C09142=1184.403,208.297,-60.136,-177.705,6.782,148.579
C09143=1184.398,208.546,-60.161,-177.703,6.784,148.579
C09144=1184.394,208.794,-60.185,-177.700,6.786,148.579
C09145=1184.389,209.044,-60.210,-177.698,6.788,148.579
C09146=1184.385,209.292,-60.234,-177.695,6.790,148.578
C09147=1184.381,209.541,-60.258,-177.692,6.792,148.578
C09148=1184.376,209.790,-60.283,-177.690,6.794,148.578
C09149=1184.372,210.039,-60.307,-177.687,6.796,148.577
C09150=1184.366,210.309,-60.333,-177.684,6.799,148.577
C09151=1184.361,210.579,-60.360,-177.681,6.801,148.577
C09152=1184.357,210.850,-60.387,-177.678,6.803,148.576
C09153=1184.351,211.121,-60.414,-177.675,6.806,148.576
C09154=1184.347,211.369,-60.438,-177.673,6.808,148.576
C09155=1184.342,211.618,-60.463,-177.670,6.810,148.576
C09156=1184.338,211.867,-60.487,-177.667,6.812,148.575
C09157=1184.333,212.116,-60.512,-177.665,6.815,148.575
C09158=1184.329,212.365,-60.536,-177.662,6.816,148.575
C09159=1184.324,212.613,-60.561,-177.659,6.818,148.575
C09160=1184.320,212.861,-60.586,-177.657,6.821,148.575
C09161=1184.315,213.111,-60.611,-177.654,6.823,148.574
C09162=1184.310,213.359,-60.635,-177.651,6.825,148.574
C09163=1184.306,213.608,-60.659,-177.649,6.827,148.574
C09164=1184.301,213.857,-60.684,-177.646,6.830,148.573
C09165=1184.297,214.106,-60.708,-177.643,6.831,148.573
C09166=1184.293,214.354,-60.734,-177.640,6.833,148.573
C09167=1184.288,214.603,-60.758,-177.638,6.835,148.573
C09168=1184.283,214.851,-60.783,-177.635,6.838,148.572
C09169=1184.279,215.101,-60.808,-177.632,6.840,148.572
C09170=1184.275,215.349,-60.833,-177.630,6.842,148.572
C09171=1184.270,215.598,-60.858,-177.627,6.845,148.572
C09172=1184.266,215.847,-60.882,-177.624,6.846,148.571
C09173=1184.260,216.095,-60.907,-177.622,6.848,148.571
C09174=1184.256,216.344,-60.932,-177.620,6.850,148.571
C09175=1184.252,216.592,-60.956,-177.616,6.853,148.570
C09176=1184.247,216.842,-60.981,-177.614,6.855,148.570
C09177=1184.243,217.090,-61.007,-177.611,6.857,148.570
C09178=1184.239,217.339,-61.031,-177.608,6.859,148.570
C09179=1184.234,217.588,-61.056,-177.606,6.862,148.570
C09180=1184.229,217.836,-61.081,-177.603,6.863,148.569
C09181=1184.225,218.085,-61.106,-177.601,6.866,148.569
C09182=1184.220,218.334,-61.130,-177.598,6.868,148.569
C09183=1184.216,218.583,-61.156,-177.595,6.870,148.569
C09184=1184.210,218.831,-61.181,-177.593,6.873,148.568
C09185=1184.207,219.080,-61.206,-177.590,6.875,148.568
C09186=1184.202,219.329,-61.231,-177.587,6.877,148.568
C09187=1184.198,219.577,-61.256,-177.585,6.879,148.568
C09188=1184.192,219.826,-61.281,-177.582,6.881,148.567
C09189=1184.189,220.075,-61.306,-177.579,6.883,148.567
C09190=1184.184,220.323,-61.331,-177.577,6.885,148.567
C09191=1184.180,220.572,-61.357,-177.574,6.888,148.567
C09192=1184.175,220.821,-61.381,-177.572,6.890,148.566
C09193=1184.171,221.069,-61.406,-177.569,6.892,148.566
C09194=1184.166,221.318,-61.431,-177.566,6.895,148.566
C09195=1184.162,221.567,-61.457,-177.564,6.897,148.566
C09196=1184.157,221.816,-61.482,-177.561,6.899,148.565
C09197=1184.152,222.064,-61.507,-177.558,6.901,148.565
C09198=1184.147,222.313,-61.532,-177.556,6.903,148.565
C09199=1184.144,222.562,-61.557,-177.553,6.905,148.565
C09200=1184.139,222.810,-61.583,-177.550,6.908,148.565
C09201=1184.134,223.059,-61.608,-177.548,6.910,148.564
C09202=1184.130,223.308,-61.633,-177.545,6.912,148.564
C09203=1184.125,223.557,-61.658,-177.542,6.915,148.564
C09204=1184.121,223.805,-61.684,-177.539,6.916,148.564
C09205=1184.116,224.054,-61.709,-177.537,6.919,148.563
C09206=1184.111,224.303,-61.734,-177.534,6.921,148.563
C09207=1184.107,224.551,-61.759,-177.531,6.923,148.563
C09208=1184.103,224.800,-61.785,-177.529,6.925,148.563
C09209=1184.099,225.048,-61.810,-177.526,6.928,148.562
C09210=1184.094,225.297,-61.835,-177.524,6.930,148.562
C09211=1184.090,225.546,-61.861,-177.521,6.932,148.562
C09212=1184.085,225.794,-61.886,-177.518,6.935,148.562
C09213=1184.080,226.043,-61.911,-177.516,6.937,148.562
C09214=1184.076,226.292,-61.937,-177.513,6.939,148.561
C09215=1184.071,226.540,-61.962,-177.510,6.941,148.561
C09216=1184.067,226.789,-61.988,-177.508,6.943,148.561
C09217=1184.063,227.038,-62.014,-177.505,6.946,148.561
C09218=1184.058,227.287,-62.039,-177.502,6.948,148.560
C09219=1184.053,227.535,-62.064,-177.500,6.950,148.560
C09220=1184.048,227.784,-62.090,-177.497,6.953,148.560
C09221=1184.044,228.032,-62.116,-177.494,6.955,148.560
C09222=1184.040,228.281,-62.141,-177.492,6.957,148.560
C09223=1184.035,228.529,-62.167,-177.489,6.959,148.559
C09224=1184.031,228.778,-62.192,-177.487,6.961,148.559
C09225=1184.027,229.027,-62.218,-177.484,6.964,148.559
C09226=1184.022,229.276,-62.243,-177.481,6.966,148.559
C09227=1184.017,229.524,-62.269,-177.479,6.968,148.558
C09228=1184.013,229.773,-62.294,-177.476,6.971,148.558
C09229=1184.008,230.021,-62.320,-177.473,6.973,148.558
C09230=1184.004,230.270,-62.345,-177.471,6.975,148.558
C09231=1183.999,230.519,-62.372,-177.468,6.978,148.558
C09232=1183.995,230.768,-62.398,-177.465,6.979,148.557
C09233=1183.990,231.016,-62.423,-177.463,6.982,148.557
C09234=1183.986,231.265,-62.449,-177.460,6.984,148.557
C09235=1183.982,231.514,-62.474,-177.458,6.986,148.557
C09236=1183.977,231.762,-62.500,-177.454,6.989,148.556
C09237=1183.973,232.011,-62.526,-177.452,6.991,148.556
C09238=1183.968,232.259,-62.551,-177.449,6.994,148.556
C09239=1183.963,232.509,-62.578,-177.447,6.996,148.556
C09240=1183.959,232.756,-62.604,-177.444,6.998,148.556
C09241=1183.955,233.005,-62.630,-177.442,7.001,148.556
C09242=1183.950,233.254,-62.655,-177.439,7.003,148.555
C09243=1183.946,233.502,-62.681,-177.436,7.006,148.555
C09244=1183.941,233.751,-62.707,-177.434,7.007,148.555
C09245=1183.936,234.000,-62.733,-177.431,7.009,148.555
C09246=1183.932,234.249,-62.758,-177.428,7.012,148.554
C09247=1183.928,234.497,-62.784,-177.426,7.014,148.554
C09248=1183.923,234.745,-62.810,-177.423,7.017,148.554
C09249=1183.919,234.994,-62.837,-177.421,7.019,148.554
C09250=1183.914,235.243,-62.862,-177.418,7.021,148.554
C09251=1183.910,235.492,-62.888,-177.415,7.024,148.554
C09252=1183.906,235.740,-62.914,-177.413,7.026,148.553
C09253=1183.901,235.988,-62.941,-177.410,7.029,148.553
C09254=1183.896,236.260,-62.969,-177.407,7.031,148.553
C09255=1183.891,236.531,-62.997,-177.404,7.033,148.553
C09256=1183.886,236.804,-63.026,-177.401,7.036,148.552
C09257=1183.882,237.075,-63.055,-177.398,7.039,148.552
C09258=1183.877,237.323,-63.080,-177.396,7.041,148.552
C09259=1183.873,237.572,-63.106,-177.393,7.044,148.552
C09260=1183.868,237.820,-63.133,-177.390,7.046,148.552
C09261=1183.864,238.069,-63.159,-177.388,7.048,148.552
C09262=1183.860,238.318,-63.185,-177.385,7.050,148.551
C09263=1183.855,238.566,-63.212,-177.383,7.053,148.551
C09264=1183.851,238.815,-63.237,-177.380,7.055,148.551
C09265=1183.845,239.064,-63.263,-177.377,7.057,148.551
C09266=1183.841,239.312,-63.290,-177.375,7.060,148.551
C09267=1183.837,239.561,-63.316,-177.372,7.062,148.550
C09268=1183.832,239.809,-63.343,-177.369,7.065,148.550
C09269=1183.828,240.058,-63.368,-177.367,7.067,148.550
C09270=1183.823,240.306,-63.395,-177.364,7.070,148.550
C09271=1183.819,240.555,-63.421,-177.361,7.072,148.550
C09272=1183.815,240.804,-63.447,-177.359,7.074,148.550
C09273=1183.810,241.052,-63.474,-177.356,7.077,148.549
C09274=1183.805,241.301,-63.499,-177.354,7.079,148.549
C09275=1183.801,241.549,-63.526,-177.351,7.082,148.549
C09276=1183.797,241.798,-63.552,-177.348,7.084,148.549
C09277=1183.792,242.046,-63.579,-177.346,7.087,148.549
C09278=1183.788,242.294,-63.606,-177.343,7.088,148.548
C09279=1183.783,242.544,-63.632,-177.340,7.091,148.548
C09280=1183.779,242.792,-63.659,-177.338,7.093,148.548
C09281=1183.774,243.041,-63.685,-177.335,7.096,148.548
C09282=1183.770,243.289,-63.711,-177.333,7.098,148.548
C09283=1183.765,243.538,-63.738,-177.330,7.101,148.548
C09284=1183.761,243.786,-63.764,-177.327,7.103,148.547
C09285=1183.757,244.035,-63.791,-177.325,7.106,148.547
C09286=1183.752,244.284,-63.817,-177.322,7.108,148.547
C09287=1183.748,244.532,-63.844,-177.319,7.111,148.547
C09288=1183.744,244.780,-63.870,-177.317,7.113,148.547
C09289=1183.739,245.030,-63.897,-177.314,7.115,148.547
C09290=1183.735,245.278,-63.923,-177.312,7.118,148.547
C09291=1183.730,245.526,-63.950,-177.309,7.120,148.546
C09292=1183.726,245.775,-63.977,-177.306,7.123,148.546
C09293=1183.721,246.023,-64.003,-177.304,7.125,148.546
C09294=1183.717,246.272,-64.030,-177.301,7.127,148.546
C09295=1183.713,246.520,-64.057,-177.299,7.130,148.546
C09296=1183.708,246.769,-64.084,-177.296,7.132,148.546
C09297=1183.703,247.018,-64.110,-177.293,7.134,148.545
C09298=1183.699,247.266,-64.137,-177.291,7.137,148.545
C09299=1183.695,247.514,-64.164,-177.288,7.139,148.545
C09300=1183.690,247.763,-64.191,-177.285,7.142,148.545
C09301=1183.686,248.011,-64.217,-177.283,7.144,148.545
C09302=1183.681,248.260,-64.243,-177.280,7.147,148.545
C09303=1183.677,248.509,-64.271,-177.278,7.149,148.544
C09304=1183.673,248.757,-64.297,-177.275,7.152,148.544
C09305=1183.668,249.005,-64.324,-177.272,7.155,148.544
C09306=1183.663,249.254,-64.351,-177.270,7.157,148.544
C09307=1183.659,249.502,-64.378,-177.267,7.160,148.544
C09308=1183.655,249.751,-64.405,-177.264,7.162,148.544
C09309=1183.650,249.999,-64.432,-177.261,7.165,148.544
C09310=1183.646,250.247,-64.458,-177.259,7.167,148.543
C09311=1183.642,250.497,-64.485,-177.256,7.169,148.543
C09312=1183.637,250.746,-64.512,-177.254,7.172,148.543
C09313=1183.632,250.994,-64.539,-177.251,7.175,148.543
C09314=1183.629,251.242,-64.566,-177.249,7.176,148.543
C09315=1183.624,251.491,-64.593,-177.246,7.179,148.543
C09316=1183.619,251.739,-64.620,-177.244,7.182,148.543
C09317=1183.615,251.988,-64.647,-177.241,7.184,148.542
C09318=1183.610,252.236,-64.674,-177.238,7.186,148.542
C09319=1183.607,252.485,-64.701,-177.236,7.189,148.542
C09320=1183.602,252.733,-64.728,-177.233,7.191,148.542
C09321=1183.598,252.982,-64.755,-177.230,7.194,148.542
C09322=1183.593,253.230,-64.782,-177.227,7.197,148.542
C09323=1183.588,253.479,-64.810,-177.225,7.199,148.542
C09324=1183.584,253.727,-64.837,-177.222,7.202,148.541
C09325=1183.580,253.975,-64.863,-177.220,7.204,148.541
C09326=1183.576,254.224,-64.890,-177.217,7.207,148.541
C09327=1183.571,254.473,-64.918,-177.215,7.209,148.541
C09328=1183.567,254.721,-64.945,-177.212,7.212,148.541
C09329=1183.562,254.969,-64.972,-177.210,7.214,148.541
C09330=1183.557,255.218,-64.999,-177.207,7.217,148.541
C09331=1183.553,255.466,-65.027,-177.204,7.220,148.541
C09332=1183.549,255.715,-65.054,-177.202,7.222,148.540
C09333=1183.544,255.963,-65.082,-177.199,7.225,148.540
C09334=1183.540,256.211,-65.108,-177.197,7.227,148.540
C09335=1183.536,256.460,-65.135,-177.193,7.230,148.540
C09336=1183.532,256.709,-65.163,-177.191,7.232,148.540
C09337=1183.527,256.957,-65.190,-177.189,7.235,148.540
C09338=1183.523,257.206,-65.218,-177.186,7.238,148.540
C09339=1183.518,257.454,-65.245,-177.183,7.240,148.539
C09340=1183.513,257.703,-65.272,-177.180,7.242,148.539
C09341=1183.510,257.951,-65.300,-177.178,7.245,148.539
C09342=1183.505,258.200,-65.327,-177.176,7.248,148.539
C09343=1183.500,258.448,-65.354,-177.173,7.249,148.539
C09344=1183.496,258.696,-65.382,-177.170,7.252,148.539
C09345=1183.492,258.945,-65.409,-177.167,7.255,148.539
C09346=1183.487,259.193,-65.437,-177.165,7.258,148.539
C09347=1183.483,259.442,-65.464,-177.163,7.261,148.539
C09348=1183.479,259.691,-65.491,-177.160,7.262,148.538
C09349=1183.474,259.939,-65.519,-177.157,7.265,148.538
C09350=1183.470,260.187,-65.546,-177.154,7.268,148.538
C09351=1183.465,260.435,-65.574,-177.152,7.270,148.538
C09352=1183.461,260.685,-65.602,-177.149,7.273,148.538
C09353=1183.456,260.932,-65.630,-177.147,7.275,148.538
C09354=1183.452,261.181,-65.657,-177.144,7.278,148.538
C09355=1183.448,261.429,-65.685,-177.141,7.281,148.538
C09356=1183.443,261.678,-65.712,-177.139,7.283,148.538
C09357=1183.439,261.926,-65.740,-177.136,7.286,148.537
C09358=1183.434,262.199,-65.771,-177.133,7.289,148.537
C09359=1183.429,262.472,-65.801,-177.131,7.292,148.537
C09360=1183.425,262.745,-65.831,-177.127,7.295,148.537
C09361=1183.420,263.017,-65.861,-177.125,7.298,148.537
C09362=1183.416,263.267,-65.889,-177.123,7.300,148.537
C09363=1183.411,263.515,-65.917,-177.120,7.303,148.537
C09364=1183.406,263.763,-65.944,-177.117,7.305,148.536
C09365=1183.402,264.012,-65.972,-177.114,7.308,148.536
C09366=1183.398,264.260,-66.000,-177.112,7.311,148.536
C09367=1183.394,264.509,-66.027,-177.110,7.313,148.536
C09368=1183.389,264.757,-66.056,-177.107,7.316,148.536
C09369=1183.384,265.005,-66.084,-177.104,7.319,148.536
C09370=1183.380,265.254,-66.111,-177.101,7.321,148.536
C09371=1183.376,265.502,-66.139,-177.099,7.324,148.536
C09372=1183.372,265.750,-66.167,-177.096,7.327,148.536
C09373=1183.367,265.999,-66.195,-177.094,7.329,148.536
C09374=1183.362,266.247,-66.222,-177.091,7.332,148.536
C09375=1183.359,266.496,-66.250,-177.089,7.334,148.536
C09376=1183.354,266.744,-66.279,-177.086,7.337,148.535
C09377=1183.349,266.992,-66.307,-177.083,7.339,148.535
C09378=1183.345,267.241,-66.334,-177.081,7.342,148.535
C09379=1183.341,267.489,-66.362,-177.078,7.345,148.535
C09380=1183.336,267.738,-66.391,-177.075,7.348,148.535
C09381=1183.332,267.986,-66.418,-177.073,7.350,148.535
C09382=1183.328,268.234,-66.447,-177.070,7.353,148.535
C09383=1183.323,268.483,-66.474,-177.067,7.355,148.535
C09384=1183.319,268.732,-66.502,-177.065,7.358,148.535
C09385=1183.315,268.980,-66.530,-177.062,7.361,148.535
C09386=1183.310,269.228,-66.558,-177.060,7.364,148.534
C09387=1183.306,269.476,-66.587,-177.057,7.366,148.534
C09388=1183.302,269.724,-66.614,-177.055,7.369,148.534
C09389=1183.297,269.973,-66.643,-177.052,7.372,148.534
C09390=1183.293,270.221,-66.671,-177.049,7.374,148.534
C09391=1183.288,270.470,-66.700,-177.047,7.377,148.534
C09392=1183.284,270.718,-66.727,-177.044,7.379,148.534
C09393=1183.280,270.966,-66.756,-177.042,7.382,148.534
C09394=1183.275,271.215,-66.784,-177.039,7.385,148.534
C09395=1183.271,271.463,-66.812,-177.036,7.388,148.534
C09396=1183.266,271.711,-66.840,-177.034,7.390,148.534
C09397=1183.262,271.960,-66.869,-177.031,7.393,148.534
C09398=1183.257,272.208,-66.897,-177.029,7.396,148.534
C09399=1183.254,272.457,-66.925,-177.026,7.398,148.533
C09400=1183.249,272.706,-66.954,-177.023,7.401,148.533
C09401=1183.245,272.953,-66.982,-177.021,7.404,148.533
C09402=1183.240,273.202,-67.010,-177.018,7.406,148.533
C09403=1183.236,273.450,-67.038,-177.016,7.409,148.533
C09404=1183.232,273.699,-67.066,-177.013,7.412,148.533
C09405=1183.227,273.947,-67.095,-177.011,7.414,148.533
C09406=1183.223,274.195,-67.124,-177.008,7.417,148.533
C09407=1183.219,274.443,-67.152,-177.005,7.420,148.533
C09408=1183.214,274.692,-67.181,-177.003,7.422,148.533
C09409=1183.210,274.941,-67.209,-177.000,7.425,148.533
C09410=1183.205,275.189,-67.237,-176.998,7.428,148.533
C09411=1183.202,275.437,-67.266,-176.995,7.431,148.532
C09412=1183.197,275.685,-67.294,-176.992,7.433,148.532
C09413=1183.193,275.933,-67.322,-176.990,7.436,148.532
C09414=1183.188,276.182,-67.351,-176.987,7.439,148.532
C09415=1183.183,276.431,-67.380,-176.985,7.441,148.532
C09416=1183.180,276.679,-67.408,-176.982,7.444,148.532
C09417=1183.175,276.927,-67.437,-176.979,7.447,148.532
C09418=1183.171,277.175,-67.465,-176.977,7.449,148.532
C09419=1183.167,277.424,-67.494,-176.974,7.452,148.532
C09420=1183.162,277.672,-67.523,-176.972,7.455,148.532
C09421=1183.158,277.920,-67.551,-176.969,7.458,148.532
C09422=1183.154,278.169,-67.580,-176.967,7.460,148.532
C09423=1183.150,278.416,-67.608,-176.964,7.463,148.532
C09424=1183.145,278.665,-67.637,-176.961,7.466,148.532
C09425=1183.141,278.914,-67.666,-176.959,7.468,148.532
C09426=1183.137,279.161,-67.694,-176.956,7.471,148.532
C09427=1183.132,279.410,-67.724,-176.954,7.474,148.532
C09428=1183.128,279.659,-67.752,-176.951,7.477,148.532
C09429=1183.123,279.907,-67.781,-176.949,7.479,148.531
C09430=1183.119,280.155,-67.810,-176.946,7.482,148.531
C09431=1183.115,280.404,-67.838,-176.943,7.485,148.531
C09432=1183.111,280.652,-67.868,-176.940,7.488,148.531
C09433=1183.106,280.900,-67.896,-176.938,7.490,148.531
C09434=1183.102,281.148,-67.925,-176.935,7.493,148.531
C09435=1183.098,281.397,-67.954,-176.933,7.496,148.531
C09436=1183.093,281.645,-67.983,-176.930,7.498,148.531
C09437=1183.088,281.893,-68.012,-176.928,7.501,148.531
C09438=1183.085,282.141,-68.040,-176.925,7.504,148.531
C09439=1183.081,282.390,-68.070,-176.922,7.507,148.531
C09440=1183.076,282.638,-68.098,-176.920,7.510,148.531
C09441=1183.071,282.886,-68.128,-176.917,7.513,148.531
C09442=1183.067,283.135,-68.156,-176.915,7.515,148.531
C09443=1183.064,283.383,-68.185,-176.912,7.518,148.531
C09444=1183.059,283.630,-68.214,-176.910,7.521,148.531
C09445=1183.054,283.879,-68.243,-176.907,7.524,148.531
C09446=1183.050,284.128,-68.273,-176.904,7.527,148.530
C09447=1183.046,284.377,-68.301,-176.902,7.530,148.530
C09448=1183.041,284.624,-68.330,-176.899,7.532,148.530
C09449=1183.037,284.872,-68.360,-176.897,7.535,148.530
C09450=1183.033,285.120,-68.389,-176.894,7.538,148.531
C09451=1183.029,285.369,-68.417,-176.892,7.541,148.531
C09452=1183.025,285.617,-68.447,-176.890,7.543,148.530
C09453=1183.020,285.865,-68.476,-176.887,7.546,148.530
C09454=1183.015,286.114,-68.505,-176.884,7.549,148.530
C09455=1183.011,286.362,-68.534,-176.881,7.552,148.530
C09456=1183.007,286.610,-68.564,-176.879,7.555,148.530
C09457=1183.003,286.859,-68.593,-176.877,7.557,148.530
C09458=1182.998,287.106,-68.622,-176.874,7.560,148.530
C09459=1182.993,287.355,-68.651,-176.871,7.563,148.530
C09460=1182.989,287.603,-68.680,-176.868,7.566,148.530
C09461=1182.985,287.852,-68.710,-176.866,7.568,148.530
C09462=1182.981,288.125,-68.742,-176.863,7.572,148.530
C09463=1182.976,288.401,-68.775,-176.860,7.575,148.530
C09464=1182.971,288.675,-68.806,-176.857,7.578,148.530
C09465=1182.966,288.950,-68.840,-176.855,7.581,148.530
C09466=1182.962,289.198,-68.869,-176.852,7.584,148.530
C09467=1182.958,289.447,-68.899,-176.849,7.587,148.530
C09468=1182.954,289.695,-68.928,-176.847,7.589,148.530
C09469=1182.949,289.942,-68.957,-176.844,7.592,148.530
C09470=1182.944,290.191,-68.986,-176.842,7.595,148.530
C09471=1182.940,290.440,-69.015,-176.839,7.598,148.530
C09472=1182.936,290.688,-69.045,-176.836,7.601,148.530
C09473=1182.932,290.936,-69.074,-176.834,7.604,148.530
C09474=1182.928,291.184,-69.104,-176.831,7.607,148.530
C09475=1182.924,291.432,-69.134,-176.829,7.610,148.530
C09476=1182.920,291.680,-69.163,-176.826,7.613,148.530
C09477=1182.915,291.928,-69.193,-176.824,7.615,148.530
C09478=1182.911,292.177,-69.223,-176.822,7.618,148.530
C09479=1182.906,292.425,-69.252,-176.819,7.621,148.530
C09480=1182.902,292.674,-69.282,-176.816,7.624,148.530
C09481=1182.898,292.922,-69.311,-176.813,7.627,148.530
C09482=1182.894,293.170,-69.341,-176.811,7.629,148.530
C09483=1182.889,293.418,-69.370,-176.808,7.632,148.529
C09484=1182.885,293.666,-69.399,-176.806,7.635,148.529
C09485=1182.880,293.914,-69.430,-176.803,7.638,148.529
C09486=1182.876,294.162,-69.459,-176.801,7.641,148.530
C09487=1182.872,294.410,-69.489,-176.799,7.644,148.530
C09488=1182.868,294.659,-69.518,-176.796,7.647,148.530
C09489=1182.863,294.907,-69.548,-176.793,7.650,148.530
C09490=1182.859,295.155,-69.579,-176.790,7.653,148.529
C09491=1182.855,295.403,-69.608,-176.788,7.656,148.529
C09492=1182.851,295.651,-69.637,-176.785,7.659,148.529
C09493=1182.846,295.900,-69.667,-176.783,7.661,148.529
C09494=1182.842,296.148,-69.698,-176.781,7.664,148.530
C09495=1182.838,296.396,-69.727,-176.778,7.667,148.530
C09496=1182.833,296.644,-69.757,-176.775,7.670,148.529
C09497=1182.829,296.892,-69.787,-176.772,7.673,148.529
C09498=1182.825,297.141,-69.817,-176.770,7.675,148.529
C09499=1182.821,297.389,-69.847,-176.768,7.678,148.529
C09500=1182.817,297.637,-69.877,-176.765,7.681,148.529
C09501=1182.813,297.885,-69.906,-176.763,7.685,148.530
C09502=1182.808,298.134,-69.936,-176.760,7.687,148.530
C09503=1182.804,298.382,-69.966,-176.757,7.690,148.529
C09504=1182.800,298.630,-69.996,-176.755,7.693,148.529
C09505=1182.795,298.878,-70.027,-176.752,7.696,148.529
C09506=1182.791,299.126,-70.056,-176.750,7.699,148.529
C09507=1182.787,299.374,-70.086,-176.747,7.702,148.530
C09508=1182.782,299.622,-70.116,-176.745,7.705,148.530
C09509=1182.778,299.871,-70.146,-176.742,7.708,148.530
C09510=1182.774,300.119,-70.177,-176.740,7.710,148.529
C09511=1182.769,300.367,-70.206,-176.737,7.713,148.529
C09512=1182.766,300.615,-70.237,-176.734,7.716,148.529
C09513=1182.761,300.864,-70.267,-176.732,7.719,148.530
C09514=1182.757,301.111,-70.297,-176.729,7.722,148.530
C09515=1182.752,301.360,-70.327,-176.727,7.725,148.530
C09516=1182.749,301.608,-70.357,-176.724,7.728,148.529
C09517=1182.744,301.856,-70.388,-176.722,7.731,148.529
C09518=1182.740,302.104,-70.417,-176.719,7.734,148.530
C09519=1182.736,302.351,-70.447,-176.717,7.737,148.530
C09520=1182.732,302.601,-70.478,-176.714,7.740,148.530
C09521=1182.728,302.848,-70.508,-176.711,7.743,148.530
C09522=1182.723,303.096,-70.539,-176.709,7.746,148.530
C09523=1182.719,303.345,-70.568,-176.707,7.748,148.530
C09524=1182.714,303.593,-70.599,-176.704,7.751,148.530
C09525=1182.710,303.840,-70.629,-176.701,7.754,148.530
C09526=1182.705,304.089,-70.659,-176.699,7.757,148.530
C09527=1182.701,304.337,-70.690,-176.696,7.760,148.530
C09528=1182.698,304.585,-70.720,-176.694,7.764,148.530
C09529=1182.693,304.833,-70.751,-176.691,7.767,148.530
C09530=1182.689,305.081,-70.781,-176.689,7.769,148.530
C09531=1182.684,305.329,-70.811,-176.686,7.772,148.530
C09532=1182.681,305.578,-70.842,-176.684,7.775,148.530
C09533=1182.676,305.826,-70.873,-176.681,7.778,148.530
C09534=1182.672,306.074,-70.902,-176.678,7.781,148.530
C09535=1182.667,306.322,-70.933,-176.676,7.784,148.530
C09536=1182.663,306.570,-70.964,-176.673,7.787,148.530
C09537=1182.660,306.818,-70.994,-176.671,7.790,148.530
C09538=1182.655,307.066,-71.025,-176.669,7.793,148.530
C09539=1182.650,307.314,-71.056,-176.666,7.796,148.530
C09540=1182.646,307.562,-71.085,-176.664,7.799,148.530
C09541=1182.642,307.811,-71.116,-176.661,7.802,148.530
C09542=1182.638,308.059,-71.147,-176.658,7.805,148.530
C09543=1182.634,308.307,-71.177,-176.655,7.808,148.530
C09544=1182.629,308.555,-71.208,-176.653,7.811,148.530
C09545=1182.625,308.803,-71.239,-176.651,7.813,148.530
C09546=1182.621,309.051,-71.269,-176.648,7.816,148.530
C09547=1182.617,309.299,-71.300,-176.646,7.820,148.530
C09548=1182.612,309.547,-71.331,-176.643,7.823,148.530
C09549=1182.609,309.795,-71.361,-176.641,7.826,148.530
C09550=1182.604,310.043,-71.392,-176.638,7.829,148.530
C09551=1182.599,310.291,-71.423,-176.636,7.832,148.531
C09552=1182.595,310.540,-71.454,-176.633,7.835,148.531
C09553=1182.592,310.787,-71.484,-176.631,7.837,148.530
C09554=1182.587,311.035,-71.515,-176.628,7.840,148.531
C09555=1182.583,311.284,-71.546,-176.626,7.843,148.531
C09556=1182.578,311.532,-71.577,-176.623,7.846,148.531
C09557=1182.574,311.780,-71.607,-176.621,7.850,148.531
C09558=1182.570,312.028,-71.638,-176.618,7.853,148.531
C09559=1182.566,312.276,-71.669,-176.615,7.856,148.531
C09560=1182.562,312.524,-71.700,-176.613,7.859,148.531
C09561=1182.557,312.772,-71.732,-176.610,7.862,148.531
C09562=1182.554,313.020,-71.762,-176.608,7.864,148.531
C09563=1182.549,313.268,-71.792,-176.606,7.868,148.531
C09564=1182.545,313.516,-71.824,-176.603,7.871,148.531
C09565=1182.541,313.764,-71.855,-176.601,7.874,148.531
C09566=1182.536,314.041,-71.889,-176.598,7.877,148.531
C09567=1182.531,314.318,-71.924,-176.595,7.881,148.531
C09568=1182.527,314.593,-71.959,-176.592,7.884,148.531
C09569=1182.522,314.871,-71.992,-176.589,7.888,148.531
C09570=1182.518,315.118,-72.024,-176.587,7.890,148.532
C09571=1182.514,315.367,-72.055,-176.585,7.893,148.532
C09572=1182.509,315.615,-72.086,-176.582,7.896,148.532
C09573=1182.505,315.863,-72.117,-176.580,7.899,148.532
C09574=1182.501,316.111,-72.148,-176.577,7.902,148.532
C09575=1182.497,316.359,-72.180,-176.575,7.906,148.532
C09576=1182.492,316.607,-72.210,-176.572,7.909,148.532
C09577=1182.488,316.855,-72.242,-176.569,7.912,148.532
C09578=1182.484,317.103,-72.273,-176.567,7.915,148.532
C09579=1182.480,317.351,-72.304,-176.564,7.918,148.532
C09580=1182.476,317.599,-72.336,-176.561,7.921,148.532
C09581=1182.471,317.847,-72.366,-176.560,7.923,148.532
C09582=1182.467,318.095,-72.398,-176.557,7.926,148.532
C09583=1182.463,318.343,-72.429,-176.555,7.930,148.532
C09584=1182.459,318.591,-72.461,-176.552,7.933,148.532
C09585=1182.454,318.839,-72.492,-176.549,7.936,148.532
C09586=1182.451,319.087,-72.523,-176.547,7.939,148.533
C09587=1182.446,319.335,-72.554,-176.544,7.942,148.533
C09588=1182.442,319.583,-72.586,-176.542,7.945,148.533
C09589=1182.438,319.831,-72.617,-176.539,7.948,148.533
C09590=1182.434,320.079,-72.649,-176.537,7.952,148.533
C09591=1182.429,320.327,-72.679,-176.534,7.955,148.533
C09592=1182.426,320.575,-72.711,-176.532,7.958,148.533
C09593=1182.421,320.823,-72.743,-176.529,7.961,148.533
C09594=1182.417,321.071,-72.774,-176.527,7.963,148.533
C09595=1182.413,321.318,-72.805,-176.525,7.966,148.533
C09596=1182.409,321.567,-72.836,-176.522,7.969,148.533
C09597=1182.405,321.814,-72.868,-176.520,7.973,148.534
C09598=1182.401,322.063,-72.900,-176.517,7.976,148.534
C09599=1182.396,322.310,-72.931,-176.515,7.979,148.534
C09600=1182.392,322.559,-72.963,-176.512,7.982,148.534
C09601=1182.388,322.806,-72.994,-176.510,7.985,148.534
C09602=1182.384,323.055,-73.026,-176.507,7.988,148.534
C09603=1182.380,323.303,-73.057,-176.505,7.992,148.534
C09604=1182.376,323.550,-73.089,-176.502,7.995,148.534
C09605=1182.372,323.799,-73.120,-176.500,7.998,148.534
C09606=1182.366,324.047,-73.152,-176.497,8.001,148.534
C09607=1182.363,324.295,-73.184,-176.495,8.004,148.535
C09608=1182.359,324.543,-73.216,-176.493,8.007,148.535
C09609=1182.355,324.790,-73.247,-176.491,8.010,148.535
C09610=1182.351,325.039,-73.278,-176.488,8.013,148.535
C09611=1182.346,325.286,-73.310,-176.486,8.016,148.535
C09612=1182.342,325.534,-73.342,-176.483,8.019,148.535
C09613=1182.338,325.782,-73.374,-176.481,8.022,148.535
C09614=1182.334,326.030,-73.406,-176.478,8.025,148.535
C09615=1182.330,326.278,-73.438,-176.476,8.029,148.535
C09616=1182.325,326.526,-73.469,-176.473,8.032,148.535
C09617=1182.321,326.774,-73.501,-176.471,8.035,148.535
C09618=1182.318,327.022,-73.533,-176.468,8.038,148.535
C09619=1182.312,327.270,-73.565,-176.466,8.041,148.536
C09620=1182.309,327.518,-73.596,-176.464,8.045,148.536
C09621=1182.305,327.766,-73.628,-176.461,8.048,148.536
C09622=1182.300,328.013,-73.660,-176.459,8.051,148.536
C09623=1182.296,328.261,-73.692,-176.456,8.054,148.536
C09624=1182.293,328.510,-73.724,-176.454,8.057,148.536
C09625=1182.288,328.757,-73.756,-176.451,8.060,148.536
C09626=1182.284,329.005,-73.788,-176.449,8.064,148.536
C09627=1182.280,329.253,-73.820,-176.447,8.067,148.537
C09628=1182.275,329.501,-73.852,-176.444,8.070,148.537
C09629=1182.271,329.749,-73.884,-176.442,8.072,148.537
C09630=1182.268,329.997,-73.916,-176.439,8.075,148.537
C09631=1182.263,330.245,-73.948,-176.437,8.079,148.537
C09632=1182.259,330.493,-73.980,-176.435,8.082,148.537
C09633=1182.254,330.741,-74.012,-176.432,8.085,148.537
C09634=1182.251,330.989,-74.044,-176.430,8.088,148.537
C09635=1182.246,331.236,-74.077,-176.428,8.092,148.538
C09636=1182.242,331.484,-74.108,-176.425,8.095,148.538
C09637=1182.239,331.732,-74.140,-176.423,8.098,148.538
C09638=1182.234,331.980,-74.172,-176.420,8.101,148.538
C09639=1182.230,332.228,-74.204,-176.418,8.104,148.538
C09640=1182.225,332.476,-74.237,-176.415,8.108,148.538
C09641=1182.222,332.724,-74.269,-176.413,8.111,148.538
C09642=1182.217,332.971,-74.301,-176.410,8.114,148.539
C09643=1182.213,333.219,-74.333,-176.408,8.117,148.539
C09644=1182.209,333.468,-74.366,-176.405,8.120,148.539
C09645=1182.205,333.715,-74.398,-176.403,8.124,148.539
C09646=1182.201,333.963,-74.431,-176.401,8.127,148.539
C09647=1182.197,334.211,-74.462,-176.399,8.130,148.539
C09648=1182.192,334.459,-74.495,-176.396,8.133,148.539
C09649=1182.189,334.707,-74.527,-176.394,8.137,148.540
C09650=1182.184,334.955,-74.560,-176.391,8.140,148.540
C09651=1182.180,335.203,-74.592,-176.389,8.143,148.540
C09652=1182.176,335.450,-74.624,-176.386,8.146,148.540
C09653=1182.172,335.698,-74.657,-176.384,8.150,148.540
C09654=1182.168,335.946,-74.689,-176.382,8.153,148.540
C09655=1182.164,336.194,-74.722,-176.379,8.156,148.540
C09656=1182.160,336.442,-74.753,-176.377,8.159,148.541
C09657=1182.155,336.689,-74.786,-176.375,8.162,148.541
C09658=1182.151,336.937,-74.819,-176.372,8.166,148.541
C09659=1182.147,337.185,-74.851,-176.370,8.169,148.541
C09660=1182.143,337.433,-74.884,-176.368,8.172,148.541
C09661=1182.139,337.681,-74.917,-176.365,8.175,148.542
C09662=1182.135,337.929,-74.949,-176.363,8.179,148.542
C09663=1182.131,338.177,-74.981,-176.360,8.182,148.542
C09664=1182.126,338.424,-75.014,-176.358,8.185,148.542
C09665=1182.123,338.672,-75.046,-176.356,8.188,148.542
C09666=1182.118,338.920,-75.079,-176.354,8.192,148.542
C09667=1182.114,339.168,-75.112,-176.351,8.195,148.543
C09668=1182.110,339.416,-75.144,-176.349,8.198,148.543
C09669=1182.106,339.664,-75.177,-176.346,8.201,148.543
C09670=1182.102,339.942,-75.214,-176.344,8.205,148.543
C09671=1182.096,340.222,-75.250,-176.341,8.209,148.543
C09672=1182.092,340.501,-75.287,-176.339,8.212,148.543
C09673=1182.087,340.780,-75.324,-176.336,8.216,148.544
C09674=1182.084,341.027,-75.357,-176.333,8.219,148.544
C09675=1182.079,341.276,-75.389,-176.331,8.223,148.544
C09676=1182.075,341.523,-75.422,-176.329,8.226,148.544
C09677=1182.071,341.771,-75.455,-176.327,8.229,148.544
C09678=1182.067,342.019,-75.487,-176.324,8.232,148.545
C09679=1182.062,342.266,-75.520,-176.322,8.236,148.545
C09680=1182.058,342.514,-75.553,-176.320,8.239,148.545
C09681=1182.054,342.762,-75.586,-176.318,8.242,148.545
C09682=1182.050,343.010,-75.619,-176.315,8.246,148.545
C09683=1182.046,343.258,-75.652,-176.313,8.249,148.546
C09684=1182.042,343.505,-75.685,-176.310,8.252,148.546
C09685=1182.038,343.753,-75.718,-176.308,8.255,148.546
C09686=1182.034,344.001,-75.750,-176.306,8.259,148.546
C09687=1182.030,344.249,-75.783,-176.304,8.262,148.546
C09688=1182.025,344.497,-75.816,-176.301,8.265,148.547
C09689=1182.021,344.744,-75.850,-176.299,8.269,148.547
C09690=1182.017,344.992,-75.883,-176.297,8.272,148.547
C09691=1182.013,345.240,-75.916,-176.295,8.275,148.547
C09692=1182.009,345.488,-75.948,-176.292,8.279,148.547
C09693=1182.005,345.736,-75.981,-176.290,8.282,148.548
C09694=1182.001,345.983,-76.014,-176.288,8.285,148.548
C09695=1181.997,346.231,-76.047,-176.285,8.288,148.548
C09696=1181.993,346.479,-76.080,-176.283,8.292,148.548
C09697=1181.989,346.726,-76.114,-176.281,8.295,148.549
C09698=1181.984,346.974,-76.147,-176.279,8.298,148.549
C09699=1181.980,347.222,-76.180,-176.276,8.302,148.549
C09700=1181.976,347.470,-76.213,-176.274,8.305,148.549
C09701=1181.972,347.717,-76.246,-176.272,8.308,148.549
C09702=1181.968,347.965,-76.279,-176.270,8.312,148.550
C09703=1181.964,348.213,-76.313,-176.267,8.315,148.550
C09704=1181.960,348.461,-76.346,-176.266,8.319,148.550
C09705=1181.956,348.709,-76.379,-176.263,8.322,148.550
C09706=1181.952,348.957,-76.412,-176.261,8.325,148.551
C09707=1181.948,349.204,-76.446,-176.259,8.329,148.551
C09708=1181.944,349.452,-76.479,-176.257,8.332,148.551
C09709=1181.940,349.700,-76.512,-176.254,8.335,148.551
C09710=1181.935,349.948,-76.545,-176.252,8.339,148.552
C09711=1181.932,350.195,-76.579,-176.250,8.342,148.552
C09712=1181.927,350.442,-76.612,-176.247,8.345,148.552
C09713=1181.923,350.690,-76.645,-176.246,8.349,148.552
C09714=1181.918,350.938,-76.679,-176.243,8.352,148.553
C09715=1181.914,351.186,-76.712,-176.241,8.355,148.553
C09716=1181.911,351.434,-76.746,-176.239,8.359,148.553
C09717=1181.907,351.682,-76.779,-176.237,8.362,148.553
C09718=1181.903,351.929,-76.813,-176.234,8.366,148.554
C09719=1181.899,352.177,-76.846,-176.232,8.370,148.554
C09720=1181.894,352.425,-76.879,-176.230,8.373,148.554
C09721=1181.891,352.672,-76.913,-176.227,8.376,148.554
C09722=1181.886,352.920,-76.947,-176.225,8.380,148.555
C09723=1181.882,353.168,-76.980,-176.223,8.383,148.555
C09724=1181.878,353.416,-77.013,-176.221,8.387,148.555
C09725=1181.874,353.663,-77.047,-176.219,8.390,148.556
C09726=1181.870,353.911,-77.080,-176.217,8.393,148.556
C09727=1181.866,354.159,-77.113,-176.215,8.397,148.556
C09728=1181.861,354.406,-77.148,-176.213,8.400,148.556
C09729=1181.858,354.654,-77.181,-176.210,8.404,148.557
C09730=1181.854,354.902,-77.215,-176.208,8.407,148.557
C09731=1181.850,355.149,-77.248,-176.206,8.410,148.557
C09732=1181.846,355.397,-77.282,-176.204,8.414,148.558
C09733=1181.841,355.644,-77.316,-176.202,8.417,148.558
C09734=1181.838,355.893,-77.350,-176.200,8.421,148.558
C09735=1181.834,356.140,-77.383,-176.198,8.424,148.558
C09736=1181.830,356.388,-77.417,-176.195,8.427,148.559
C09737=1181.825,356.636,-77.450,-176.194,8.431,148.559
C09738=1181.822,356.884,-77.485,-176.191,8.435,148.559
C09739=1181.817,357.131,-77.518,-176.189,8.439,148.560
C09740=1181.814,357.378,-77.552,-176.187,8.442,148.560
C09741=1181.809,357.626,-77.585,-176.184,8.445,148.560
C09742=1181.806,357.874,-77.620,-176.183,8.449,148.561
C09743=1181.801,358.122,-77.653,-176.180,8.452,148.561
C09744=1181.797,358.369,-77.687,-176.178,8.456,148.561
C09745=1181.793,358.616,-77.721,-176.176,8.459,148.562
C09746=1181.789,358.865,-77.755,-176.174,8.463,148.562
C09747=1181.785,359.112,-77.789,-176.172,8.466,148.562
C09748=1181.781,359.360,-77.822,-176.170,8.470,148.563
C09749=1181.777,359.607,-77.856,-176.168,8.473,148.563
C09750=1181.773,359.855,-77.891,-176.166,8.477,148.563
C09751=1181.769,360.103,-77.924,-176.164,8.480,148.563
C09752=1181.765,360.350,-77.958,-176.162,8.484,148.564
C09753=1181.761,360.598,-77.993,-176.160,8.487,148.564
C09754=1181.757,360.846,-78.026,-176.158,8.491,148.565
C09755=1181.752,361.093,-78.060,-176.156,8.494,148.565
C09756=1181.749,361.341,-78.095,-176.154,8.498,148.565
C09757=1181.745,361.589,-78.128,-176.152,8.501,148.566
C09758=1181.740,361.836,-78.162,-176.150,8.505,148.566
C09759=1181.737,362.084,-78.197,-176.148,8.508,148.566
C09760=1181.733,362.332,-78.231,-176.146,8.512,148.567
C09761=1181.728,362.579,-78.264,-176.144,8.515,148.567
C09762=1181.724,362.827,-78.299,-176.142,8.519,148.567
C09763=1181.721,363.075,-78.333,-176.140,8.522,148.568
C09764=1181.716,363.322,-78.367,-176.139,8.526,148.568
C09765=1181.713,363.570,-78.402,-176.137,8.529,148.569
C09766=1181.708,363.818,-78.435,-176.134,8.533,148.569
C09767=1181.705,364.066,-78.470,-176.133,8.536,148.569
C09768=1181.700,364.313,-78.504,-176.131,8.540,148.570
C09769=1181.696,364.560,-78.538,-176.129,8.544,148.570
C09770=1181.692,364.808,-78.573,-176.128,8.546,148.571
C09771=1181.688,365.055,-78.607,-176.126,8.550,148.571
C09772=1181.684,365.303,-78.641,-176.124,8.554,148.571
C09773=1181.681,365.551,-78.675,-176.122,8.557,148.572
C09774=1181.675,365.833,-78.714,-176.120,8.562,148.572
C09775=1181.671,366.114,-78.753,-176.118,8.565,148.573
C09776=1181.666,366.396,-78.792,-176.116,8.569,148.573
C09777=1181.662,366.677,-78.831,-176.114,8.573,148.574
C09778=1181.658,366.925,-78.866,-176.112,8.577,148.574
C09779=1181.655,367.172,-78.900,-176.110,8.581,148.575
C09780=1181.650,367.420,-78.934,-176.109,8.583,148.575
C09781=1181.646,367.667,-78.968,-176.107,8.587,148.575
C09782=1181.642,367.915,-79.003,-176.105,8.591,148.576
C09783=1181.638,368.162,-79.038,-176.104,8.594,148.576
C09784=1181.634,368.410,-79.072,-176.102,8.598,148.577
C09785=1181.630,368.658,-79.106,-176.100,8.602,148.577
C09786=1181.626,368.906,-79.141,-176.099,8.605,148.578
C09787=1181.622,369.153,-79.175,-176.097,8.608,148.578
C09788=1181.618,369.401,-79.210,-176.095,8.612,148.579
C09789=1181.613,369.648,-79.244,-176.094,8.616,148.579
C09790=1181.611,369.896,-79.279,-176.093,8.619,148.580
C09791=1181.606,370.143,-79.314,-176.091,8.622,148.580
C09792=1181.601,370.391,-79.348,-176.089,8.626,148.580
C09793=1181.598,370.638,-79.382,-176.087,8.629,148.581
C09794=1181.594,370.886,-79.417,-176.087,8.633,148.581
C09795=1181.590,371.134,-79.452,-176.085,8.636,148.582
C09796=1181.586,371.380,-79.486,-176.083,8.640,148.582
C09797=1181.582,371.628,-79.521,-176.082,8.643,148.583
C09798=1181.578,371.876,-79.556,-176.080,8.647,148.583
C09799=1181.574,372.124,-79.590,-176.078,8.650,148.584
C09800=1181.570,372.371,-79.624,-176.078,8.653,148.584
C09801=1181.566,372.619,-79.660,-176.076,8.657,148.585
C09802=1181.562,372.866,-79.694,-176.074,8.661,148.585
C09803=1181.558,373.114,-79.729,-176.073,8.664,148.586
C09804=1181.554,373.362,-79.763,-176.072,8.667,148.586
C09805=1181.550,373.609,-79.799,-176.070,8.671,148.587
C09806=1181.546,373.857,-79.833,-176.069,8.674,148.587
C09807=1181.542,374.104,-79.868,-176.067,8.678,148.588
C09808=1181.539,374.351,-79.903,-176.067,8.681,148.588
C09809=1181.534,374.599,-79.937,-176.065,8.685,148.589
C09810=1181.530,374.847,-79.972,-176.063,8.688,148.590
C09811=1181.526,375.094,-80.007,-176.062,8.692,148.590
C09812=1181.522,375.342,-80.042,-176.061,8.695,148.591
C09813=1181.518,375.589,-80.076,-176.060,8.698,148.591
C09814=1181.514,375.837,-80.111,-176.058,8.702,148.592
C09815=1181.510,376.085,-80.146,-176.057,8.705,148.592
C09816=1181.506,376.332,-80.181,-176.056,8.709,148.593
C09817=1181.502,376.580,-80.216,-176.055,8.712,148.593
C09818=1181.498,376.827,-80.251,-176.054,8.715,148.594
C09819=1181.494,377.075,-80.286,-176.052,8.719,148.594
C09820=1181.490,377.322,-80.320,-176.052,8.722,148.595
C09821=1181.486,377.569,-80.356,-176.050,8.725,148.595
C09822=1181.482,377.817,-80.391,-176.049,8.729,148.596
C09823=1181.478,378.065,-80.425,-176.048,8.732,148.597
C09824=1181.474,378.312,-80.461,-176.047,8.736,148.597
C09825=1181.470,378.560,-80.495,-176.046,8.739,148.598
C09826=1181.466,378.807,-80.531,-176.045,8.743,148.598
C09827=1181.462,379.055,-80.565,-176.043,8.745,148.599
C09828=1181.458,379.302,-80.601,-176.042,8.748,148.599
C09829=1181.454,379.550,-80.635,-176.041,8.752,148.600
C09830=1181.450,379.797,-80.670,-176.040,8.755,148.601
C09831=1181.447,380.044,-80.706,-176.039,8.759,148.601
C09832=1181.443,380.292,-80.740,-176.039,8.762,148.602
C09833=1181.438,380.539,-80.776,-176.037,8.766,148.602
C09834=1181.434,380.787,-80.810,-176.036,8.769,148.603
C09835=1181.431,381.035,-80.846,-176.036,8.772,148.604
C09836=1181.426,381.282,-80.880,-176.035,8.775,148.604
C09837=1181.422,381.530,-80.916,-176.034,8.778,148.605
C09838=1181.419,381.777,-80.952,-176.033,8.782,148.605
C09839=1181.414,382.025,-80.986,-176.032,8.785,148.606
C09840=1181.411,382.272,-81.022,-176.031,8.788,148.607
C09841=1181.407,382.520,-81.056,-176.030,8.791,148.607
C09842=1181.402,382.767,-81.092,-176.029,8.794,148.608
C09843=1181.399,383.014,-81.127,-176.028,8.797,148.608
C09844=1181.394,383.262,-81.162,-176.028,8.800,148.609
C09845=1181.390,383.509,-81.197,-176.027,8.804,148.610
C09846=1181.387,383.757,-81.233,-176.026,8.807,148.610
C09847=1181.382,384.004,-81.267,-176.026,8.810,148.611
C09848=1181.379,384.252,-81.303,-176.025,8.813,148.611
C09849=1181.375,384.499,-81.338,-176.024,8.816,148.612
C09850=1181.371,384.747,-81.373,-176.024,8.820,148.613
C09851=1181.367,384.994,-81.408,-176.023,8.823,148.613
C09852=1181.363,385.242,-81.444,-176.022,8.826,148.614
C09853=1181.359,385.489,-81.479,-176.021,8.829,148.614
C09854=1181.355,385.737,-81.514,-176.020,8.832,148.615
C09855=1181.351,385.984,-81.549,-176.020,8.835,148.616
C09856=1181.347,386.232,-81.585,-176.020,8.838,148.616
C09857=1181.342,386.479,-81.620,-176.019,8.841,148.617
C09858=1181.338,386.727,-81.656,-176.018,8.844,148.618
C09859=1181.335,386.974,-81.691,-176.018,8.847,148.618
C09860=1181.331,387.222,-81.727,-176.017,8.850,148.619
C09861=1181.327,387.469,-81.762,-176.017,8.853,148.620
C09862=1181.323,387.717,-81.797,-176.016,8.856,148.620
C09863=1181.319,387.964,-81.832,-176.015,8.859,148.621
C09864=1181.315,388.211,-81.867,-176.015,8.862,148.622
C09865=1181.311,388.459,-81.903,-176.015,8.865,148.622
C09866=1181.308,388.706,-81.938,-176.014,8.868,148.623
C09867=1181.304,388.954,-81.973,-176.014,8.870,148.623
C09868=1181.299,389.201,-82.008,-176.013,8.873,148.624
C09869=1181.295,389.449,-82.045,-176.013,8.877,148.625
C09870=1181.291,389.696,-82.080,-176.013,8.879,148.625
C09871=1181.288,389.944,-82.116,-176.012,8.883,148.626
C09872=1181.283,390.191,-82.151,-176.012,8.885,148.627
C09873=1181.280,390.438,-82.186,-176.012,8.888,148.627
C09874=1181.276,390.686,-82.221,-176.011,8.890,148.628
C09875=1181.272,390.934,-82.257,-176.011,8.894,148.629
C09876=1181.268,391.181,-82.292,-176.011,8.896,148.629
C09877=1181.263,391.428,-82.328,-176.010,8.899,148.630
C09878=1181.259,391.712,-82.369,-176.009,8.903,148.631
C09879=1181.255,391.996,-82.409,-176.009,8.906,148.631
C09880=1181.251,392.280,-82.450,-176.009,8.909,148.632
C09881=1181.246,392.565,-82.491,-176.009,8.912,148.633
C09882=1181.241,392.812,-82.526,-176.009,8.915,148.634
C09883=1181.238,393.059,-82.562,-176.008,8.918,148.634
C09884=1181.234,393.307,-82.597,-176.008,8.920,148.635
C09885=1181.230,393.554,-82.633,-176.008,8.923,148.635
C09886=1181.226,393.802,-82.669,-176.008,8.926,148.636
C09887=1181.222,394.049,-82.704,-176.007,8.928,148.637
C09888=1181.218,394.296,-82.740,-176.008,8.931,148.637
C09889=1181.214,394.544,-82.775,-176.007,8.934,148.638
C09890=1181.211,394.791,-82.811,-176.007,8.936,148.639
C09891=1181.205,395.039,-82.846,-176.007,8.939,148.639
C09892=1181.202,395.286,-82.882,-176.006,8.942,148.640
C09893=1181.198,395.534,-82.917,-176.006,8.944,148.640
C09894=1181.194,395.781,-82.953,-176.006,8.947,148.641
C09895=1181.191,396.029,-82.988,-176.006,8.949,148.642
C09896=1181.186,396.276,-83.024,-176.006,8.952,148.642
C09897=1181.182,396.524,-83.060,-176.006,8.954,148.643
C09898=1181.178,396.771,-83.095,-176.006,8.957,148.644
C09899=1181.175,397.019,-83.131,-176.006,8.960,148.644
C09900=1181.170,397.266,-83.167,-176.005,8.962,148.645
C09901=1181.166,397.513,-83.202,-176.006,8.965,148.646
C09902=1181.163,397.760,-83.238,-176.005,8.967,148.646
C09903=1181.159,398.008,-83.274,-176.006,8.970,148.647
C09904=1181.155,398.255,-83.310,-176.005,8.972,148.647
C09905=1181.151,398.503,-83.345,-176.005,8.974,148.648
C09906=1181.147,398.750,-83.381,-176.005,8.977,148.649
C09907=1181.143,398.997,-83.416,-176.005,8.979,148.649
C09908=1181.139,399.245,-83.452,-176.005,8.981,148.650
C09909=1181.135,399.492,-83.488,-176.005,8.984,148.651
C09910=1181.131,399.740,-83.523,-176.005,8.986,148.651
C09911=1181.127,399.987,-83.559,-176.005,8.989,148.652
C09912=1181.123,400.235,-83.595,-176.005,8.991,148.653
C09913=1181.119,400.482,-83.630,-176.005,8.994,148.653
C09914=1181.115,400.730,-83.666,-176.005,8.996,148.654
C09915=1181.112,400.977,-83.701,-176.005,8.999,148.654
C09916=1181.107,401.224,-83.737,-176.005,9.001,148.655
C09917=1181.103,401.472,-83.773,-176.005,9.003,148.656
C09918=1181.100,401.719,-83.809,-176.005,9.006,148.656
C09919=1181.095,401.966,-83.845,-176.005,9.008,148.657
C09920=1181.092,402.214,-83.881,-176.005,9.011,148.658
C09921=1181.088,402.461,-83.916,-176.005,9.013,148.658
C09922=1181.084,402.708,-83.951,-176.005,9.016,148.659
C09923=1181.079,402.956,-83.988,-176.005,9.018,148.659
C09924=1181.076,403.204,-84.023,-176.005,9.020,148.660
C09925=1181.072,403.451,-84.059,-176.005,9.022,148.661
C09926=1181.068,403.698,-84.096,-176.005,9.024,148.661
C09927=1181.064,403.946,-84.131,-176.005,9.027,148.662
C09928=1181.060,404.192,-84.166,-176.005,9.029,148.662
C09929=1181.056,404.440,-84.202,-176.005,9.032,148.663
C09930=1181.052,404.688,-84.238,-176.005,9.033,148.663
C09931=1181.048,404.935,-84.273,-176.005,9.036,148.664
C09932=1181.045,405.183,-84.309,-176.005,9.038,148.665
C09933=1181.041,405.430,-84.346,-176.005,9.040,148.665
C09934=1181.037,405.677,-84.381,-176.006,9.042,148.666
C09935=1181.033,405.924,-84.417,-176.005,9.044,148.666
C09936=1181.028,406.172,-84.453,-176.005,9.047,148.667
C09937=1181.025,406.420,-84.488,-176.005,9.049,148.668
C09938=1181.021,406.667,-84.524,-176.006,9.051,148.668
C09939=1181.017,406.914,-84.561,-176.006,9.053,148.669
C09940=1181.013,407.162,-84.596,-176.005,9.055,148.669
C09941=1181.009,407.409,-84.632,-176.006,9.057,148.670
C09942=1181.004,407.656,-84.668,-176.006,9.059,148.671
C09943=1181.001,407.904,-84.703,-176.006,9.062,148.671
C09944=1180.997,408.151,-84.739,-176.006,9.064,148.672
C09945=1180.993,408.399,-84.776,-176.006,9.065,148.672
C09946=1180.989,408.646,-84.811,-176.006,9.068,148.673
C09947=1180.986,408.894,-84.847,-176.006,9.070,148.673
C09948=1180.981,409.141,-84.883,-176.006,9.072,148.674
C09949=1180.978,409.388,-84.919,-176.006,9.074,148.675
C09950=1180.973,409.635,-84.955,-176.007,9.076,148.675
C09951=1180.969,409.883,-84.990,-176.006,9.078,148.676
C09952=1180.966,410.130,-85.026,-176.007,9.081,148.676
C09953=1180.962,410.378,-85.063,-176.007,9.082,148.677
C09954=1180.958,410.625,-85.098,-176.007,9.084,148.677
C09955=1180.954,410.873,-85.134,-176.007,9.087,148.678
C09956=1180.950,411.120,-85.170,-176.007,9.088,148.679
C09957=1180.946,411.367,-85.206,-176.007,9.091,148.679
C09958=1180.942,411.614,-85.241,-176.007,9.092,148.679
C09959=1180.938,411.862,-85.278,-176.007,9.095,148.680
C09960=1180.934,412.109,-85.313,-176.008,9.096,148.681
C09961=1180.930,412.357,-85.350,-176.007,9.098,148.681
C09962=1180.926,412.604,-85.386,-176.007,9.100,148.682
C09963=1180.923,412.852,-85.421,-176.008,9.102,148.682
C09964=1180.918,413.099,-85.457,-176.008,9.104,148.683
C09965=1180.915,413.346,-85.494,-176.008,9.106,148.683
C09966=1180.911,413.594,-85.530,-176.008,9.108,148.684
C09967=1180.906,413.841,-85.565,-176.008,9.110,148.684
C09968=1180.903,414.088,-85.601,-176.008,9.112,148.685
C09969=1180.899,414.336,-85.637,-176.008,9.114,148.685
C09970=1180.895,414.583,-85.673,-176.008,9.116,148.686
C09971=1180.890,414.831,-85.709,-176.008,9.117,148.686
C09972=1180.887,415.078,-85.745,-176.008,9.120,148.687
C09973=1180.883,415.325,-85.781,-176.008,9.121,148.687
C09974=1180.879,415.552,-85.814,-176.008,9.123,148.688
C09975=1180.876,415.779,-85.847,-176.008,9.125,148.688
C09976=1180.874,416.006,-85.879,-176.008,9.127,148.689
C09977=1180.872,416.234,-85.913,-176.008,9.128,148.689
C09978=1180.872,416.460,-85.945,-176.009,9.130,148.690
C09979=1180.872,416.687,-85.978,-176.009,9.131,148.690
C09980=1180.874,416.914,-86.010,-176.009,9.134,148.691
C09981=1180.877,417.141,-86.043,-176.009,9.135,148.691
C09982=1180.455,417.142,-86.085,-176.012,9.146,148.695
C09983=1180.452,416.914,-86.053,-176.012,9.144,148.694
C09984=1180.451,416.686,-86.021,-176.012,9.142,148.694
C09985=1180.451,416.457,-85.987,-176.012,9.141,148.693
C09986=1180.451,416.229,-85.954,-176.012,9.139,148.693
C09987=1180.453,416.000,-85.922,-176.012,9.138,148.693
C09988=1180.454,415.771,-85.888,-176.012,9.136,148.692
C09989=1180.458,415.542,-85.855,-176.012,9.134,148.692
C09990=1180.462,415.313,-85.822,-176.012,9.132,148.691
C09991=1180.466,415.067,-85.786,-176.011,9.131,148.691
C09992=1180.470,414.820,-85.750,-176.011,9.128,148.690
C09993=1180.474,414.572,-85.714,-176.011,9.127,148.690
C09994=1180.477,414.325,-85.678,-176.011,9.124,148.689
C09995=1180.482,414.077,-85.642,-176.011,9.123,148.689
C09996=1180.485,413.830,-85.606,-176.011,9.121,148.688
//INST
///DATE 2021/06/15 17:24
///ATTR SC,RW,RJ
////FRAME ROBOT
///GROUP1 RB1
NOP
MOVL C00000 V=800.0 PL=0
MOVL C00001 V=800.0 PL=0
MOVL C00002 V=800.0 PL=0
MOVL C00003 V=800.0 PL=0
MOVL C00004 V=800.0 PL=0
MOVL C00005 V=800.0 PL=0
MOVL C00006 V=800.0 PL=0
MOVL C00007 V=800.0 PL=0
MOVL C00008 V=800.0 PL=0
MOVL C00009 V=800.0 PL=0
MOVL C00010 V=800.0 PL=0
MOVL C00011 V=800.0 PL=0
MOVL C00012 V=800.0 PL=0
MOVL C00013 V=800.0 PL=0
MOVL C00014 V=800.0 PL=0
MOVL C00015 V=800.0 PL=0
MOVL C00016 V=800.0 PL=0
MOVL C00017 V=800.0 PL=0
MOVL C00018 V=800.0 PL=0
MOVL C00019 V=800.0 PL=0
MOVL C00020 V=800.0 PL=0
MOVL C00021 V=800.0 PL=0
MOVL C00022 V=800.0 PL=0
MOVL C00023 V=800.0 PL=0
MOVL C00024 V=800.0 PL=0
MOVL C00025 V=800.0 PL=0
MOVL C00026 V=800.0 PL=0
MOVL C00027 V=800.0 PL=0
MOVL C00028 V=800.0 PL=0
MOVL C00029 V=800.0 PL=0
MOVL C00030 V=800.0 PL=0
MOVL C00031 V=800.0 PL=0
MOVL C00032 V=800.0 PL=0
MOVL C00033 V=800.0 PL=0
MOVL C00034 V=800.0 PL=0
MOVL C00035 V=800.0 PL=0
MOVL C00036 V=800.0 PL=0
MOVL C00037 V=800.0 PL=0
MOVL C00038 V=800.0 PL=0
MOVL C00039 V=800.0 PL=0
MOVL C00040 V=800.0 PL=0
MOVL C00041 V=800.0 PL=0
MOVL C00042 V=800.0 PL=0
MOVL C00043 V=800.0 PL=0
MOVL C00044 V=800.0 PL=0
MOVL C00045 V=800.0 PL=0
MOVL C00046 V=800.0 PL=0
MOVL C00047 V=800.0 PL=0
MOVL C00048 V=800.0 PL=0
MOVL C00049 V=800.0 PL=0
MOVL C00050 V=800.0 PL=0
MOVL C00051 V=800.0 PL=0
MOVL C00052 V=800.0 PL=0
MOVL C00053 V=800.0 PL=0
MOVL C00054 V=800.0 PL=0
MOVL C00055 V=800.0 PL=0
MOVL C00056 V=800.0 PL=0
MOVL C00057 V=800.0 PL=0
MOVL C00058 V=800.0 PL=0
MOVL C00059 V=800.0 PL=0
MOVL C00060 V=800.0 PL=0
MOVL C00061 V=800.0 PL=0
MOVL C00062 V=800.0 PL=0
MOVL C00063 V=800.0 PL=0
MOVL C00064 V=800.0 PL=0
MOVL C00065 V=800.0 PL=0
MOVL C00066 V=800.0 PL=0
MOVL C00067 V=800.0 PL=0
MOVL C00068 V=800.0 PL=0
MOVL C00069 V=800.0 PL=0
MOVL C00070 V=800.0 PL=0
MOVL C00071 V=800.0 PL=0
MOVL C00072 V=800.0 PL=0
MOVL C00073 V=800.0 PL=0
MOVL C00074 V=800.0 PL=0
MOVL C00075 V=800.0 PL=0
MOVL C00076 V=800.0 PL=0
MOVL C00077 V=800.0 PL=0
MOVL C00078 V=800.0 PL=0
MOVL C00079 V=800.0 PL=0
MOVL C00080 V=800.0 PL=0
MOVL C00081 V=800.0 PL=0
MOVL C00082 V=800.0 PL=0
MOVL C00083 V=800.0 PL=0
MOVL C00084 V=800.0 PL=0
MOVL C00085 V=800.0 PL=0
MOVL C00086 V=800.0 PL=0
MOVL C00087 V=800.0 PL=0
MOVL C00088 V=800.0 PL=0
MOVL C00089 V=800.0 PL=0
MOVL C00090 V=800.0 PL=0
MOVL C00091 V=800.0 PL=0
MOVL C00092 V=800.0 PL=0
MOVL C00093 V=800.0 PL=0
MOVL C00094 V=800.0 PL=0
MOVL C00095 V=800.0 PL=0
MOVL C00096 V=800.0 PL=0
MOVL C00097 V=800.0 PL=0
MOVL C00098 V=800.0 PL=0
MOVL C00099 V=800.0 PL=0
MOVL C00100 V=800.0 PL=0
MOVL C00101 V=800.0 PL=0
MOVL C00102 V=800.0 PL=0
MOVL C00103 V=800.0 PL=0
MOVL C00104 V=800.0 PL=0
MOVL C00105 V=800.0 PL=0
MOVL C00106 V=800.0 PL=0
MOVL C00107 V=800.0 PL=0
MOVL C00108 V=800.0 PL=0
MOVL C00109 V=800.0 PL=0
MOVL C00110 V=800.0 PL=0
MOVL C00111 V=800.0 PL=0
MOVL C00112 V=800.0 PL=0
MOVL C00113 V=800.0 PL=0
MOVL C00114 V=800.0 PL=0
MOVL C00115 V=800.0 PL=0
MOVL C00116 V=800.0 PL=0
MOVL C00117 V=800.0 PL=0
MOVL C00118 V=800.0 PL=0
MOVL C00119 V=800.0 PL=0
MOVL C00120 V=800.0 PL=0
MOVL C00121 V=800.0 PL=0
MOVL C00122 V=800.0 PL=0
MOVL C00123 V=800.0 PL=0
MOVL C00124 V=800.0 PL=0
MOVL C00125 V=800.0 PL=0
MOVL C00126 V=800.0 PL=0
MOVL C00127 V=800.0 PL=0
MOVL C00128 V=800.0 PL=0
MOVL C00129 V=800.0 PL=0
MOVL C00130 V=800.0 PL=0
MOVL C00131 V=800.0 PL=0
MOVL C00132 V=800.0 PL=0
MOVL C00133 V=800.0 PL=0
MOVL C00134 V=800.0 PL=0
MOVL C00135 V=800.0 PL=0
MOVL C00136 V=800.0 PL=0
MOVL C00137 V=800.0 PL=0
MOVL C00138 V=800.0 PL=0
MOVL C00139 V=800.0 PL=0
MOVL C00140 V=800.0 PL=0
MOVL C00141 V=800.0 PL=0
MOVL C00142 V=800.0 PL=0
MOVL C00143 V=800.0 PL=0
MOVL C00144 V=800.0 PL=0
MOVL C00145 V=800.0 PL=0
MOVL C00146 V=800.0 PL=0
MOVL C00147 V=800.0 PL=0
MOVL C00148 V=800.0 PL=0
MOVL C00149 V=800.0 PL=0
MOVL C00150 V=800.0 PL=0
MOVL C00151 V=800.0 PL=0
MOVL C00152 V=800.0 PL=0
MOVL C00153 V=800.0 PL=0
MOVL C00154 V=800.0 PL=0
MOVL C00155 V=800.0 PL=0
MOVL C00156 V=800.0 PL=0
MOVL C00157 V=800.0 PL=0
MOVL C00158 V=800.0 PL=0
MOVL C00159 V=800.0 PL=0
MOVL C00160 V=800.0 PL=0
MOVL C00161 V=800.0 PL=0
MOVL C00162 V=800.0 PL=0
MOVL C00163 V=800.0 PL=0
MOVL C00164 V=800.0 PL=0
MOVL C00165 V=800.0 PL=0
MOVL C00166 V=800.0 PL=0
MOVL C00167 V=800.0 PL=0
MOVL C00168 V=800.0 PL=0
MOVL C00169 V=800.0 PL=0
MOVL C00170 V=800.0 PL=0
MOVL C00171 V=800.0 PL=0
MOVL C00172 V=800.0 PL=0
MOVL C00173 V=800.0 PL=0
MOVL C00174 V=800.0 PL=0
MOVL C00175 V=800.0 PL=0
MOVL C00176 V=800.0 PL=0
MOVL C00177 V=800.0 PL=0
MOVL C00178 V=800.0 PL=0
MOVL C00179 V=800.0 PL=0
MOVL C00180 V=800.0 PL=0
MOVL C00181 V=800.0 PL=0
MOVL C00182 V=800.0 PL=0
MOVL C00183 V=800.0 PL=0
MOVL C00184 V=800.0 PL=0
MOVL C00185 V=800.0 PL=0
MOVL C00186 V=800.0 PL=0
MOVL C00187 V=800.0 PL=0
MOVL C00188 V=800.0 PL=0
MOVL C00189 V=800.0 PL=0
MOVL C00190 V=800.0 PL=0
MOVL C00191 V=800.0 PL=0
MOVL C00192 V=800.0 PL=0
MOVL C00193 V=800.0 PL=0
MOVL C00194 V=800.0 PL=0
MOVL C00195 V=800.0 PL=0
MOVL C00196 V=800.0 PL=0
MOVL C00197 V=800.0 PL=0
MOVL C00198 V=800.0 PL=0
MOVL C00199 V=800.0 PL=0
MOVL C00200 V=800.0 PL=0
MOVL C00201 V=800.0 PL=0
MOVL C00202 V=800.0 PL=0
MOVL C00203 V=800.0 PL=0
MOVL C00204 V=800.0 PL=0
MOVL C00205 V=800.0 PL=0
MOVL C00206 V=800.0 PL=0
MOVL C00207 V=800.0 PL=0
MOVL C00208 V=800.0 PL=0
MOVL C00209 V=800.0 PL=0
MOVL C00210 V=800.0 PL=0
MOVL C00211 V=800.0 PL=0
MOVL C00212 V=800.0 PL=0
MOVL C00213 V=800.0 PL=0
MOVL C00214 V=800.0 PL=0
MOVL C00215 V=800.0 PL=0
MOVL C00216 V=800.0 PL=0
MOVL C00217 V=800.0 PL=0
MOVL C00218 V=800.0 PL=0
MOVL C00219 V=800.0 PL=0
MOVL C00220 V=800.0 PL=0
MOVL C00221 V=800.0 PL=0
MOVL C00222 V=800.0 PL=0
MOVL C00223 V=800.0 PL=0
MOVL C00224 V=800.0 PL=0
MOVL C00225 V=800.0 PL=0
MOVL C00226 V=800.0 PL=0
MOVL C00227 V=800.0 PL=0
MOVL C00228 V=800.0 PL=0
MOVL C00229 V=800.0 PL=0
MOVL C00230 V=800.0 PL=0
MOVL C00231 V=800.0 PL=0
MOVL C00232 V=800.0 PL=0
MOVL C00233 V=800.0 PL=0
MOVL C00234 V=800.0 PL=0
MOVL C00235 V=800.0 PL=0
MOVL C00236 V=800.0 PL=0
MOVL C00237 V=800.0 PL=0
MOVL C00238 V=800.0 PL=0
MOVL C00239 V=800.0 PL=0
MOVL C00240 V=800.0 PL=0
MOVL C00241 V=800.0 PL=0
MOVL C00242 V=800.0 PL=0
MOVL C00243 V=800.0 PL=0
MOVL C00244 V=800.0 PL=0
MOVL C00245 V=800.0 PL=0
MOVL C00246 V=800.0 PL=0
MOVL C00247 V=800.0 PL=0
MOVL C00248 V=800.0 PL=0
MOVL C00249 V=800.0 PL=0
MOVL C00250 V=800.0 PL=0
MOVL C00251 V=800.0 PL=0
MOVL C00252 V=800.0 PL=0
MOVL C00253 V=800.0 PL=0
MOVL C00254 V=800.0 PL=0
MOVL C00255 V=800.0 PL=0
MOVL C00256 V=800.0 PL=0
MOVL C00257 V=800.0 PL=0
MOVL C00258 V=800.0 PL=0
MOVL C00259 V=800.0 PL=0
MOVL C00260 V=800.0 PL=0
MOVL C00261 V=800.0 PL=0
MOVL C00262 V=800.0 PL=0
MOVL C00263 V=800.0 PL=0
MOVL C00264 V=800.0 PL=0
MOVL C00265 V=800.0 PL=0
MOVL C00266 V=800.0 PL=0
MOVL C00267 V=800.0 PL=0
MOVL C00268 V=800.0 PL=0
MOVL C00269 V=800.0 PL=0
MOVL C00270 V=800.0 PL=0
MOVL C00271 V=800.0 PL=0
MOVL C00272 V=800.0 PL=0
MOVL C00273 V=800.0 PL=0
MOVL C00274 V=800.0 PL=0
MOVL C00275 V=800.0 PL=0
MOVL C00276 V=800.0 PL=0
MOVL C00277 V=800.0 PL=0
MOVL C00278 V=800.0 PL=0
MOVL C00279 V=800.0 PL=0
MOVL C00280 V=800.0 PL=0
MOVL C00281 V=800.0 PL=0
MOVL C00282 V=800.0 PL=0
MOVL C00283 V=800.0 PL=0
MOVL C00284 V=800.0 PL=0
MOVL C00285 V=800.0 PL=0
MOVL C00286 V=800.0 PL=0
MOVL C00287 V=800.0 PL=0
MOVL C00288 V=800.0 PL=0
MOVL C00289 V=800.0 PL=0
MOVL C00290 V=800.0 PL=0
MOVL C00291 V=800.0 PL=0
MOVL C00292 V=800.0 PL=0
MOVL C00293 V=800.0 PL=0
MOVL C00294 V=800.0 PL=0
MOVL C00295 V=800.0 PL=0
MOVL C00296 V=800.0 PL=0
MOVL C00297 V=800.0 PL=0
MOVL C00298 V=800.0 PL=0
MOVL C00299 V=800.0 PL=0
MOVL C00300 V=800.0 PL=0
MOVL C00301 V=800.0 PL=0
MOVL C00302 V=800.0 PL=0
MOVL C00303 V=800.0 PL=0
MOVL C00304 V=800.0 PL=0
MOVL C00305 V=800.0 PL=0
MOVL C00306 V=800.0 PL=0
MOVL C00307 V=800.0 PL=0
MOVL C00308 V=800.0 PL=0
MOVL C00309 V=800.0 PL=0
MOVL C00310 V=800.0 PL=0
MOVL C00311 V=800.0 PL=0
MOVL C00312 V=800.0 PL=0
MOVL C00313 V=800.0 PL=0
MOVL C00314 V=800.0 PL=0
MOVL C00315 V=800.0 PL=0
MOVL C00316 V=800.0 PL=0
MOVL C00317 V=800.0 PL=0
MOVL C00318 V=800.0 PL=0
MOVL C00319 V=800.0 PL=0
MOVL C00320 V=800.0 PL=0
MOVL C00321 V=800.0 PL=0
MOVL C00322 V=800.0 PL=0
MOVL C00323 V=800.0 PL=0
MOVL C00324 V=800.0 PL=0
MOVL C00325 V=800.0 PL=0
MOVL C00326 V=800.0 PL=0
MOVL C00327 V=800.0 PL=0
MOVL C00328 V=800.0 PL=0
MOVL C00329 V=800.0 PL=0
MOVL C00330 V=800.0 PL=0
MOVL C00331 V=800.0 PL=0
MOVL C00332 V=800.0 PL=0
MOVL C00333 V=800.0 PL=0
MOVL C00334 V=800.0 PL=0
MOVL C00335 V=800.0 PL=0
MOVL C00336 V=800.0 PL=0
MOVL C00337 V=800.0 PL=0
MOVL C00338 V=800.0 PL=0
MOVL C00339 V=800.0 PL=0
MOVL C00340 V=800.0 PL=0
MOVL C00341 V=800.0 PL=0
MOVL C00342 V=800.0 PL=0
MOVL C00343 V=800.0 PL=0
MOVL C00344 V=800.0 PL=0
MOVL C00345 V=800.0 PL=0
MOVL C00346 V=800.0 PL=0
MOVL C00347 V=800.0 PL=0
MOVL C00348 V=800.0 PL=0
MOVL C00349 V=800.0 PL=0
MOVL C00350 V=800.0 PL=0
MOVL C00351 V=800.0 PL=0
MOVL C00352 V=800.0 PL=0
MOVL C00353 V=800.0 PL=0
MOVL C00354 V=800.0 PL=0
MOVL C00355 V=800.0 PL=0
MOVL C00356 V=800.0 PL=0
MOVL C00357 V=800.0 PL=0
MOVL C00358 V=800.0 PL=0
MOVL C00359 V=800.0 PL=0
MOVL C00360 V=800.0 PL=0
MOVL C00361 V=800.0 PL=0
MOVL C00362 V=800.0 PL=0
MOVL C00363 V=800.0 PL=0
MOVL C00364 V=800.0 PL=0
MOVL C00365 V=800.0 PL=0
MOVL C00366 V=800.0 PL=0
MOVL C00367 V=800.0 PL=0
MOVL C00368 V=800.0 PL=0
MOVL C00369 V=800.0 PL=0
MOVL C00370 V=800.0 PL=0
MOVL C00371 V=800.0 PL=0
MOVL C00372 V=800.0 PL=0
MOVL C00373 V=800.0 PL=0
MOVL C00374 V=800.0 PL=0
MOVL C00375 V=800.0 PL=0
MOVL C00376 V=800.0 PL=0
MOVL C00377 V=800.0 PL=0
MOVL C00378 V=800.0 PL=0
MOVL C00379 V=800.0 PL=0
MOVL C00380 V=800.0 PL=0
MOVL C00381 V=800.0 PL=0
MOVL C00382 V=800.0 PL=0
MOVL C00383 V=800.0 PL=0
MOVL C00384 V=800.0 PL=0
MOVL C00385 V=800.0 PL=0
MOVL C00386 V=800.0 PL=0
MOVL C00387 V=800.0 PL=0
MOVL C00388 V=800.0 PL=0
MOVL C00389 V=800.0 PL=0
MOVL C00390 V=800.0 PL=0
MOVL C00391 V=800.0 PL=0
MOVL C00392 V=800.0 PL=0
MOVL C00393 V=800.0 PL=0
MOVL C00394 V=800.0 PL=0
MOVL C00395 V=800.0 PL=0
MOVL C00396 V=800.0 PL=0
MOVL C00397 V=800.0 PL=0
MOVL C00398 V=800.0 PL=0
MOVL C00399 V=800.0 PL=0
MOVL C00400 V=800.0 PL=0
MOVL C00401 V=800.0 PL=0
MOVL C00402 V=800.0 PL=0
MOVL C00403 V=800.0 PL=0
MOVL C00404 V=800.0 PL=0
MOVL C00405 V=800.0 PL=0
MOVL C00406 V=800.0 PL=0
MOVL C00407 V=800.0 PL=0
MOVL C00408 V=800.0 PL=0
MOVL C00409 V=800.0 PL=0
MOVL C00410 V=800.0 PL=0
MOVL C00411 V=800.0 PL=0
MOVL C00412 V=800.0 PL=0
MOVL C00413 V=800.0 PL=0
MOVL C00414 V=800.0 PL=0
MOVL C00415 V=800.0 PL=0
MOVL C00416 V=800.0 PL=0
MOVL C00417 V=800.0 PL=0
MOVL C00418 V=800.0 PL=0
MOVL C00419 V=800.0 PL=0
MOVL C00420 V=800.0 PL=0
MOVL C00421 V=800.0 PL=0
MOVL C00422 V=800.0 PL=0
MOVL C00423 V=800.0 PL=0
MOVL C00424 V=800.0 PL=0
MOVL C00425 V=800.0 PL=0
MOVL C00426 V=800.0 PL=0
MOVL C00427 V=800.0 PL=0
MOVL C00428 V=800.0 PL=0
MOVL C00429 V=800.0 PL=0
MOVL C00430 V=800.0 PL=0
MOVL C00431 V=800.0 PL=0
MOVL C00432 V=800.0 PL=0
MOVL C00433 V=800.0 PL=0
MOVL C00434 V=800.0 PL=0
MOVL C00435 V=800.0 PL=0
MOVL C00436 V=800.0 PL=0
MOVL C00437 V=800.0 PL=0
MOVL C00438 V=800.0 PL=0
MOVL C00439 V=800.0 PL=0
MOVL C00440 V=800.0 PL=0
MOVL C00441 V=800.0 PL=0
MOVL C00442 V=800.0 PL=0
MOVL C00443 V=800.0 PL=0
MOVL C00444 V=800.0 PL=0
MOVL C00445 V=800.0 PL=0
MOVL C00446 V=800.0 PL=0
MOVL C00447 V=800.0 PL=0
MOVL C00448 V=800.0 PL=0
MOVL C00449 V=800.0 PL=0
MOVL C00450 V=800.0 PL=0
MOVL C00451 V=800.0 PL=0
MOVL C00452 V=800.0 PL=0
MOVL C00453 V=800.0 PL=0
MOVL C00454 V=800.0 PL=0
MOVL C00455 V=800.0 PL=0
MOVL C00456 V=800.0 PL=0
MOVL C00457 V=800.0 PL=0
MOVL C00458 V=800.0 PL=0
MOVL C00459 V=800.0 PL=0
MOVL C00460 V=800.0 PL=0
MOVL C00461 V=800.0 PL=0
MOVL C00462 V=800.0 PL=0
MOVL C00463 V=800.0 PL=0
MOVL C00464 V=800.0 PL=0
MOVL C00465 V=800.0 PL=0
MOVL C00466 V=800.0 PL=0
MOVL C00467 V=800.0 PL=0
MOVL C00468 V=800.0 PL=0
MOVL C00469 V=800.0 PL=0
MOVL C00470 V=800.0 PL=0
MOVL C00471 V=800.0 PL=0
MOVL C00472 V=800.0 PL=0
MOVL C00473 V=800.0 PL=0
MOVL C00474 V=800.0 PL=0
MOVL C00475 V=800.0 PL=0
MOVL C00476 V=800.0 PL=0
MOVL C00477 V=800.0 PL=0
MOVL C00478 V=800.0 PL=0
MOVL C00479 V=800.0 PL=0
MOVL C00480 V=800.0 PL=0
MOVL C00481 V=800.0 PL=0
MOVL C00482 V=800.0 PL=0
MOVL C00483 V=800.0 PL=0
MOVL C00484 V=800.0 PL=0
MOVL C00485 V=800.0 PL=0
MOVL C00486 V=800.0 PL=0
MOVL C00487 V=800.0 PL=0
MOVL C00488 V=800.0 PL=0
MOVL C00489 V=800.0 PL=0
MOVL C00490 V=800.0 PL=0
MOVL C00491 V=800.0 PL=0
MOVL C00492 V=800.0 PL=0
MOVL C00493 V=800.0 PL=0
MOVL C00494 V=800.0 PL=0
MOVL C00495 V=800.0 PL=0
MOVL C00496 V=800.0 PL=0
MOVL C00497 V=800.0 PL=0
MOVL C00498 V=800.0 PL=0
MOVL C00499 V=800.0 PL=0
MOVL C00500 V=800.0 PL=0
MOVL C00501 V=800.0 PL=0
MOVL C00502 V=800.0 PL=0
MOVL C00503 V=800.0 PL=0
MOVL C00504 V=800.0 PL=0
MOVL C00505 V=800.0 PL=0
MOVL C00506 V=800.0 PL=0
MOVL C00507 V=800.0 PL=0
MOVL C00508 V=800.0 PL=0
MOVL C00509 V=800.0 PL=0
MOVL C00510 V=800.0 PL=0
MOVL C00511 V=800.0 PL=0
MOVL C00512 V=800.0 PL=0
MOVL C00513 V=800.0 PL=0
MOVL C00514 V=800.0 PL=0
MOVL C00515 V=800.0 PL=0
MOVL C00516 V=800.0 PL=0
MOVL C00517 V=800.0 PL=0
MOVL C00518 V=800.0 PL=0
MOVL C00519 V=800.0 PL=0
MOVL C00520 V=800.0 PL=0
MOVL C00521 V=800.0 PL=0
MOVL C00522 V=800.0 PL=0
MOVL C00523 V=800.0 PL=0
MOVL C00524 V=800.0 PL=0
MOVL C00525 V=800.0 PL=0
MOVL C00526 V=800.0 PL=0
MOVL C00527 V=800.0 PL=0
MOVL C00528 V=800.0 PL=0
MOVL C00529 V=800.0 PL=0
MOVL C00530 V=800.0 PL=0
MOVL C00531 V=800.0 PL=0
MOVL C00532 V=800.0 PL=0
MOVL C00533 V=800.0 PL=0
MOVL C00534 V=800.0 PL=0
MOVL C00535 V=800.0 PL=0
MOVL C00536 V=800.0 PL=0
MOVL C00537 V=800.0 PL=0
MOVL C00538 V=800.0 PL=0
MOVL C00539 V=800.0 PL=0
MOVL C00540 V=800.0 PL=0
MOVL C00541 V=800.0 PL=0
MOVL C00542 V=800.0 PL=0
MOVL C00543 V=800.0 PL=0
MOVL C00544 V=800.0 PL=0
MOVL C00545 V=800.0 PL=0
MOVL C00546 V=800.0 PL=0
MOVL C00547 V=800.0 PL=0
MOVL C00548 V=800.0 PL=0
MOVL C00549 V=800.0 PL=0
MOVL C00550 V=800.0 PL=0
MOVL C00551 V=800.0 PL=0
MOVL C00552 V=800.0 PL=0
MOVL C00553 V=800.0 PL=0
MOVL C00554 V=800.0 PL=0
MOVL C00555 V=800.0 PL=0
MOVL C00556 V=800.0 PL=0
MOVL C00557 V=800.0 PL=0
MOVL C00558 V=800.0 PL=0
MOVL C00559 V=800.0 PL=0
MOVL C00560 V=800.0 PL=0
MOVL C00561 V=800.0 PL=0
MOVL C00562 V=800.0 PL=0
MOVL C00563 V=800.0 PL=0
MOVL C00564 V=800.0 PL=0
MOVL C00565 V=800.0 PL=0
MOVL C00566 V=800.0 PL=0
MOVL C00567 V=800.0 PL=0
MOVL C00568 V=800.0 PL=0
MOVL C00569 V=800.0 PL=0
MOVL C00570 V=800.0 PL=0
MOVL C00571 V=800.0 PL=0
MOVL C00572 V=800.0 PL=0
MOVL C00573 V=800.0 PL=0
MOVL C00574 V=800.0 PL=0
MOVL C00575 V=800.0 PL=0
MOVL C00576 V=800.0 PL=0
MOVL C00577 V=800.0 PL=0
MOVL C00578 V=800.0 PL=0
MOVL C00579 V=800.0 PL=0
MOVL C00580 V=800.0 PL=0
MOVL C00581 V=800.0 PL=0
MOVL C00582 V=800.0 PL=0
MOVL C00583 V=800.0 PL=0
MOVL C00584 V=800.0 PL=0
MOVL C00585 V=800.0 PL=0
MOVL C00586 V=800.0 PL=0
MOVL C00587 V=800.0 PL=0
MOVL C00588 V=800.0 PL=0
MOVL C00589 V=800.0 PL=0
MOVL C00590 V=800.0 PL=0
MOVL C00591 V=800.0 PL=0
MOVL C00592 V=800.0 PL=0
MOVL C00593 V=800.0 PL=0
MOVL C00594 V=800.0 PL=0
MOVL C00595 V=800.0 PL=0
MOVL C00596 V=800.0 PL=0
MOVL C00597 V=800.0 PL=0
MOVL C00598 V=800.0 PL=0
MOVL C00599 V=800.0 PL=0
MOVL C00600 V=800.0 PL=0
MOVL C00601 V=800.0 PL=0
MOVL C00602 V=800.0 PL=0
MOVL C00603 V=800.0 PL=0
MOVL C00604 V=800.0 PL=0
MOVL C00605 V=800.0 PL=0
MOVL C00606 V=800.0 PL=0
MOVL C00607 V=800.0 PL=0
MOVL C00608 V=800.0 PL=0
MOVL C00609 V=800.0 PL=0
MOVL C00610 V=800.0 PL=0
MOVL C00611 V=800.0 PL=0
MOVL C00612 V=800.0 PL=0
MOVL C00613 V=800.0 PL=0
MOVL C00614 V=800.0 PL=0
MOVL C00615 V=800.0 PL=0
MOVL C00616 V=800.0 PL=0
MOVL C00617 V=800.0 PL=0
MOVL C00618 V=800.0 PL=0
MOVL C00619 V=800.0 PL=0
MOVL C00620 V=800.0 PL=0
MOVL C00621 V=800.0 PL=0
MOVL C00622 V=800.0 PL=0
MOVL C00623 V=800.0 PL=0
MOVL C00624 V=800.0 PL=0
MOVL C00625 V=800.0 PL=0
MOVL C00626 V=800.0 PL=0
MOVL C00627 V=800.0 PL=0
MOVL C00628 V=800.0 PL=0
MOVL C00629 V=800.0 PL=0
MOVL C00630 V=800.0 PL=0
MOVL C00631 V=800.0 PL=0
MOVL C00632 V=800.0 PL=0
MOVL C00633 V=800.0 PL=0
MOVL C00634 V=800.0 PL=0
MOVL C00635 V=800.0 PL=0
MOVL C00636 V=800.0 PL=0
MOVL C00637 V=800.0 PL=0
MOVL C00638 V=800.0 PL=0
MOVL C00639 V=800.0 PL=0
MOVL C00640 V=800.0 PL=0
MOVL C00641 V=800.0 PL=0
MOVL C00642 V=800.0 PL=0
MOVL C00643 V=800.0 PL=0
MOVL C00644 V=800.0 PL=0
MOVL C00645 V=800.0 PL=0
MOVL C00646 V=800.0 PL=0
MOVL C00647 V=800.0 PL=0
MOVL C00648 V=800.0 PL=0
MOVL C00649 V=800.0 PL=0
MOVL C00650 V=800.0 PL=0
MOVL C00651 V=800.0 PL=0
MOVL C00652 V=800.0 PL=0
MOVL C00653 V=800.0 PL=0
MOVL C00654 V=800.0 PL=0
MOVL C00655 V=800.0 PL=0
MOVL C00656 V=800.0 PL=0
MOVL C00657 V=800.0 PL=0
MOVL C00658 V=800.0 PL=0
MOVL C00659 V=800.0 PL=0
MOVL C00660 V=800.0 PL=0
MOVL C00661 V=800.0 PL=0
MOVL C00662 V=800.0 PL=0
MOVL C00663 V=800.0 PL=0
MOVL C00664 V=800.0 PL=0
MOVL C00665 V=800.0 PL=0
MOVL C00666 V=800.0 PL=0
MOVL C00667 V=800.0 PL=0
MOVL C00668 V=800.0 PL=0
MOVL C00669 V=800.0 PL=0
MOVL C00670 V=800.0 PL=0
MOVL C00671 V=800.0 PL=0
MOVL C00672 V=800.0 PL=0
MOVL C00673 V=800.0 PL=0
MOVL C00674 V=800.0 PL=0
MOVL C00675 V=800.0 PL=0
MOVL C00676 V=800.0 PL=0
MOVL C00677 V=800.0 PL=0
MOVL C00678 V=800.0 PL=0
MOVL C00679 V=800.0 PL=0
MOVL C00680 V=800.0 PL=0
MOVL C00681 V=800.0 PL=0
MOVL C00682 V=800.0 PL=0
MOVL C00683 V=800.0 PL=0
MOVL C00684 V=800.0 PL=0
MOVL C00685 V=800.0 PL=0
MOVL C00686 V=800.0 PL=0
MOVL C00687 V=800.0 PL=0
MOVL C00688 V=800.0 PL=0
MOVL C00689 V=800.0 PL=0
MOVL C00690 V=800.0 PL=0
MOVL C00691 V=800.0 PL=0
MOVL C00692 V=800.0 PL=0
MOVL C00693 V=800.0 PL=0
MOVL C00694 V=800.0 PL=0
MOVL C00695 V=800.0 PL=0
MOVL C00696 V=800.0 PL=0
MOVL C00697 V=800.0 PL=0
MOVL C00698 V=800.0 PL=0
MOVL C00699 V=800.0 PL=0
MOVL C00700 V=800.0 PL=0
MOVL C00701 V=800.0 PL=0
MOVL C00702 V=800.0 PL=0
MOVL C00703 V=800.0 PL=0
MOVL C00704 V=800.0 PL=0
MOVL C00705 V=800.0 PL=0
MOVL C00706 V=800.0 PL=0
MOVL C00707 V=800.0 PL=0
MOVL C00708 V=800.0 PL=0
MOVL C00709 V=800.0 PL=0
MOVL C00710 V=800.0 PL=0
MOVL C00711 V=800.0 PL=0
MOVL C00712 V=800.0 PL=0
MOVL C00713 V=800.0 PL=0
MOVL C00714 V=800.0 PL=0
MOVL C00715 V=800.0 PL=0
MOVL C00716 V=800.0 PL=0
MOVL C00717 V=800.0 PL=0
MOVL C00718 V=800.0 PL=0
MOVL C00719 V=800.0 PL=0
MOVL C00720 V=800.0 PL=0
MOVL C00721 V=800.0 PL=0
MOVL C00722 V=800.0 PL=0
MOVL C00723 V=800.0 PL=0
MOVL C00724 V=800.0 PL=0
MOVL C00725 V=800.0 PL=0
MOVL C00726 V=800.0 PL=0
MOVL C00727 V=800.0 PL=0
MOVL C00728 V=800.0 PL=0
MOVL C00729 V=800.0 PL=0
MOVL C00730 V=800.0 PL=0
MOVL C00731 V=800.0 PL=0
MOVL C00732 V=800.0 PL=0
MOVL C00733 V=800.0 PL=0
MOVL C00734 V=800.0 PL=0
MOVL C00735 V=800.0 PL=0
MOVL C00736 V=800.0 PL=0
MOVL C00737 V=800.0 PL=0
MOVL C00738 V=800.0 PL=0
MOVL C00739 V=800.0 PL=0
MOVL C00740 V=800.0 PL=0
MOVL C00741 V=800.0 PL=0
MOVL C00742 V=800.0 PL=0
MOVL C00743 V=800.0 PL=0
MOVL C00744 V=800.0 PL=0
MOVL C00745 V=800.0 PL=0
MOVL C00746 V=800.0 PL=0
MOVL C00747 V=800.0 PL=0
MOVL C00748 V=800.0 PL=0
MOVL C00749 V=800.0 PL=0
MOVL C00750 V=800.0 PL=0
MOVL C00751 V=800.0 PL=0
MOVL C00752 V=800.0 PL=0
MOVL C00753 V=800.0 PL=0
MOVL C00754 V=800.0 PL=0
MOVL C00755 V=800.0 PL=0
MOVL C00756 V=800.0 PL=0
MOVL C00757 V=800.0 PL=0
MOVL C00758 V=800.0 PL=0
MOVL C00759 V=800.0 PL=0
MOVL C00760 V=800.0 PL=0
MOVL C00761 V=800.0 PL=0
MOVL C00762 V=800.0 PL=0
MOVL C00763 V=800.0 PL=0
MOVL C00764 V=800.0 PL=0
MOVL C00765 V=800.0 PL=0
MOVL C00766 V=800.0 PL=0
MOVL C00767 V=800.0 PL=0
MOVL C00768 V=800.0 PL=0
MOVL C00769 V=800.0 PL=0
MOVL C00770 V=800.0 PL=0
MOVL C00771 V=800.0 PL=0
MOVL C00772 V=800.0 PL=0
MOVL C00773 V=800.0 PL=0
MOVL C00774 V=800.0 PL=0
MOVL C00775 V=800.0 PL=0
MOVL C00776 V=800.0 PL=0
MOVL C00777 V=800.0 PL=0
MOVL C00778 V=800.0 PL=0
MOVL C00779 V=800.0 PL=0
MOVL C00780 V=800.0 PL=0
MOVL C00781 V=800.0 PL=0
MOVL C00782 V=800.0 PL=0
MOVL C00783 V=800.0 PL=0
MOVL C00784 V=800.0 PL=0
MOVL C00785 V=800.0 PL=0
MOVL C00786 V=800.0 PL=0
MOVL C00787 V=800.0 PL=0
MOVL C00788 V=800.0 PL=0
MOVL C00789 V=800.0 PL=0
MOVL C00790 V=800.0 PL=0
MOVL C00791 V=800.0 PL=0
MOVL C00792 V=800.0 PL=0
MOVL C00793 V=800.0 PL=0
MOVL C00794 V=800.0 PL=0
MOVL C00795 V=800.0 PL=0
MOVL C00796 V=800.0 PL=0
MOVL C00797 V=800.0 PL=0
MOVL C00798 V=800.0 PL=0
MOVL C00799 V=800.0 PL=0
MOVL C00800 V=800.0 PL=0
MOVL C00801 V=800.0 PL=0
MOVL C00802 V=800.0 PL=0
MOVL C00803 V=800.0 PL=0
MOVL C00804 V=800.0 PL=0
MOVL C00805 V=800.0 PL=0
MOVL C00806 V=800.0 PL=0
MOVL C00807 V=800.0 PL=0
MOVL C00808 V=800.0 PL=0
MOVL C00809 V=800.0 PL=0
MOVL C00810 V=800.0 PL=0
MOVL C00811 V=800.0 PL=0
MOVL C00812 V=800.0 PL=0
MOVL C00813 V=800.0 PL=0
MOVL C00814 V=800.0 PL=0
MOVL C00815 V=800.0 PL=0
MOVL C00816 V=800.0 PL=0
MOVL C00817 V=800.0 PL=0
MOVL C00818 V=800.0 PL=0
MOVL C00819 V=800.0 PL=0
MOVL C00820 V=800.0 PL=0
MOVL C00821 V=800.0 PL=0
MOVL C00822 V=800.0 PL=0
MOVL C00823 V=800.0 PL=0
MOVL C00824 V=800.0 PL=0
MOVL C00825 V=800.0 PL=0
MOVL C00826 V=800.0 PL=0
MOVL C00827 V=800.0 PL=0
MOVL C00828 V=800.0 PL=0
MOVL C00829 V=800.0 PL=0
MOVL C00830 V=800.0 PL=0
MOVL C00831 V=800.0 PL=0
MOVL C00832 V=800.0 PL=0
MOVL C00833 V=800.0 PL=0
MOVL C00834 V=800.0 PL=0
MOVL C00835 V=800.0 PL=0
MOVL C00836 V=800.0 PL=0
MOVL C00837 V=800.0 PL=0
MOVL C00838 V=800.0 PL=0
MOVL C00839 V=800.0 PL=0
MOVL C00840 V=800.0 PL=0
MOVL C00841 V=800.0 PL=0
MOVL C00842 V=800.0 PL=0
MOVL C00843 V=800.0 PL=0
MOVL C00844 V=800.0 PL=0
MOVL C00845 V=800.0 PL=0
MOVL C00846 V=800.0 PL=0
MOVL C00847 V=800.0 PL=0
MOVL C00848 V=800.0 PL=0
MOVL C00849 V=800.0 PL=0
MOVL C00850 V=800.0 PL=0
MOVL C00851 V=800.0 PL=0
MOVL C00852 V=800.0 PL=0
MOVL C00853 V=800.0 PL=0
MOVL C00854 V=800.0 PL=0
MOVL C00855 V=800.0 PL=0
MOVL C00856 V=800.0 PL=0
MOVL C00857 V=800.0 PL=0
MOVL C00858 V=800.0 PL=0
MOVL C00859 V=800.0 PL=0
MOVL C00860 V=800.0 PL=0
MOVL C00861 V=800.0 PL=0
MOVL C00862 V=800.0 PL=0
MOVL C00863 V=800.0 PL=0
MOVL C00864 V=800.0 PL=0
MOVL C00865 V=800.0 PL=0
MOVL C00866 V=800.0 PL=0
MOVL C00867 V=800.0 PL=0
MOVL C00868 V=800.0 PL=0
MOVL C00869 V=800.0 PL=0
MOVL C00870 V=800.0 PL=0
MOVL C00871 V=800.0 PL=0
MOVL C00872 V=800.0 PL=0
MOVL C00873 V=800.0 PL=0
MOVL C00874 V=800.0 PL=0
MOVL C00875 V=800.0 PL=0
MOVL C00876 V=800.0 PL=0
MOVL C00877 V=800.0 PL=0
MOVL C00878 V=800.0 PL=0
MOVL C00879 V=800.0 PL=0
MOVL C00880 V=800.0 PL=0
MOVL C00881 V=800.0 PL=0
MOVL C00882 V=800.0 PL=0
MOVL C00883 V=800.0 PL=0
MOVL C00884 V=800.0 PL=0
MOVL C00885 V=800.0 PL=0
MOVL C00886 V=800.0 PL=0
MOVL C00887 V=800.0 PL=0
MOVL C00888 V=800.0 PL=0
MOVL C00889 V=800.0 PL=0
MOVL C00890 V=800.0 PL=0
MOVL C00891 V=800.0 PL=0
MOVL C00892 V=800.0 PL=0
MOVL C00893 V=800.0 PL=0
MOVL C00894 V=800.0 PL=0
MOVL C00895 V=800.0 PL=0
MOVL C00896 V=800.0 PL=0
MOVL C00897 V=800.0 PL=0
MOVL C00898 V=800.0 PL=0
MOVL C00899 V=800.0 PL=0
MOVL C00900 V=800.0 PL=0
MOVL C00901 V=800.0 PL=0
MOVL C00902 V=800.0 PL=0
MOVL C00903 V=800.0 PL=0
MOVL C00904 V=800.0 PL=0
MOVL C00905 V=800.0 PL=0
MOVL C00906 V=800.0 PL=0
MOVL C00907 V=800.0 PL=0
MOVL C00908 V=800.0 PL=0
MOVL C00909 V=800.0 PL=0
MOVL C00910 V=800.0 PL=0
MOVL C00911 V=800.0 PL=0
MOVL C00912 V=800.0 PL=0
MOVL C00913 V=800.0 PL=0
MOVL C00914 V=800.0 PL=0
MOVL C00915 V=800.0 PL=0
MOVL C00916 V=800.0 PL=0
MOVL C00917 V=800.0 PL=0
MOVL C00918 V=800.0 PL=0
MOVL C00919 V=800.0 PL=0
MOVL C00920 V=800.0 PL=0
MOVL C00921 V=800.0 PL=0
MOVL C00922 V=800.0 PL=0
MOVL C00923 V=800.0 PL=0
MOVL C00924 V=800.0 PL=0
MOVL C00925 V=800.0 PL=0
MOVL C00926 V=800.0 PL=0
MOVL C00927 V=800.0 PL=0
MOVL C00928 V=800.0 PL=0
MOVL C00929 V=800.0 PL=0
MOVL C00930 V=800.0 PL=0
MOVL C00931 V=800.0 PL=0
MOVL C00932 V=800.0 PL=0
MOVL C00933 V=800.0 PL=0
MOVL C00934 V=800.0 PL=0
MOVL C00935 V=800.0 PL=0
MOVL C00936 V=800.0 PL=0
MOVL C00937 V=800.0 PL=0
MOVL C00938 V=800.0 PL=0
MOVL C00939 V=800.0 PL=0
MOVL C00940 V=800.0 PL=0
MOVL C00941 V=800.0 PL=0
MOVL C00942 V=800.0 PL=0
MOVL C00943 V=800.0 PL=0
MOVL C00944 V=800.0 PL=0
MOVL C00945 V=800.0 PL=0
MOVL C00946 V=800.0 PL=0
MOVL C00947 V=800.0 PL=0
MOVL C00948 V=800.0 PL=0
MOVL C00949 V=800.0 PL=0
MOVL C00950 V=800.0 PL=0
MOVL C00951 V=800.0 PL=0
MOVL C00952 V=800.0 PL=0
MOVL C00953 V=800.0 PL=0
MOVL C00954 V=800.0 PL=0
MOVL C00955 V=800.0 PL=0
MOVL C00956 V=800.0 PL=0
MOVL C00957 V=800.0 PL=0
MOVL C00958 V=800.0 PL=0
MOVL C00959 V=800.0 PL=0
MOVL C00960 V=800.0 PL=0
MOVL C00961 V=800.0 PL=0
MOVL C00962 V=800.0 PL=0
MOVL C00963 V=800.0 PL=0
MOVL C00964 V=800.0 PL=0
MOVL C00965 V=800.0 PL=0
MOVL C00966 V=800.0 PL=0
MOVL C00967 V=800.0 PL=0
MOVL C00968 V=800.0 PL=0
MOVL C00969 V=800.0 PL=0
MOVL C00970 V=800.0 PL=0
MOVL C00971 V=800.0 PL=0
MOVL C00972 V=800.0 PL=0
MOVL C00973 V=800.0 PL=0
MOVL C00974 V=800.0 PL=0
MOVL C00975 V=800.0 PL=0
MOVL C00976 V=800.0 PL=0
MOVL C00977 V=800.0 PL=0
MOVL C00978 V=800.0 PL=0
MOVL C00979 V=800.0 PL=0
MOVL C00980 V=800.0 PL=0
MOVL C00981 V=800.0 PL=0
MOVL C00982 V=800.0 PL=0
MOVL C00983 V=800.0 PL=0
MOVL C00984 V=800.0 PL=0
MOVL C00985 V=800.0 PL=0
MOVL C00986 V=800.0 PL=0
MOVL C00987 V=800.0 PL=0
MOVL C00988 V=800.0 PL=0
MOVL C00989 V=800.0 PL=0
MOVL C00990 V=800.0 PL=0
MOVL C00991 V=800.0 PL=0
MOVL C00992 V=800.0 PL=0
MOVL C00993 V=800.0 PL=0
MOVL C00994 V=800.0 PL=0
MOVL C00995 V=800.0 PL=0
MOVL C00996 V=800.0 PL=0
MOVL C00997 V=800.0 PL=0
MOVL C00998 V=800.0 PL=0
MOVL C00999 V=800.0 PL=0
MOVL C01000 V=800.0 PL=0
MOVL C01001 V=800.0 PL=0
MOVL C01002 V=800.0 PL=0
MOVL C01003 V=800.0 PL=0
MOVL C01004 V=800.0 PL=0
MOVL C01005 V=800.0 PL=0
MOVL C01006 V=800.0 PL=0
MOVL C01007 V=800.0 PL=0
MOVL C01008 V=800.0 PL=0
MOVL C01009 V=800.0 PL=0
MOVL C01010 V=800.0 PL=0
MOVL C01011 V=800.0 PL=0
MOVL C01012 V=800.0 PL=0
MOVL C01013 V=800.0 PL=0
MOVL C01014 V=800.0 PL=0
MOVL C01015 V=800.0 PL=0
MOVL C01016 V=800.0 PL=0
MOVL C01017 V=800.0 PL=0
MOVL C01018 V=800.0 PL=0
MOVL C01019 V=800.0 PL=0
MOVL C01020 V=800.0 PL=0
MOVL C01021 V=800.0 PL=0
MOVL C01022 V=800.0 PL=0
MOVL C01023 V=800.0 PL=0
MOVL C01024 V=800.0 PL=0
MOVL C01025 V=800.0 PL=0
MOVL C01026 V=800.0 PL=0
MOVL C01027 V=800.0 PL=0
MOVL C01028 V=800.0 PL=0
MOVL C01029 V=800.0 PL=0
MOVL C01030 V=800.0 PL=0
MOVL C01031 V=800.0 PL=0
MOVL C01032 V=800.0 PL=0
MOVL C01033 V=800.0 PL=0
MOVL C01034 V=800.0 PL=0
MOVL C01035 V=800.0 PL=0
MOVL C01036 V=800.0 PL=0
MOVL C01037 V=800.0 PL=0
MOVL C01038 V=800.0 PL=0
MOVL C01039 V=800.0 PL=0
MOVL C01040 V=800.0 PL=0
MOVL C01041 V=800.0 PL=0
MOVL C01042 V=800.0 PL=0
MOVL C01043 V=800.0 PL=0
MOVL C01044 V=800.0 PL=0
MOVL C01045 V=800.0 PL=0
MOVL C01046 V=800.0 PL=0
MOVL C01047 V=800.0 PL=0
MOVL C01048 V=800.0 PL=0
MOVL C01049 V=800.0 PL=0
MOVL C01050 V=800.0 PL=0
MOVL C01051 V=800.0 PL=0
MOVL C01052 V=800.0 PL=0
MOVL C01053 V=800.0 PL=0
MOVL C01054 V=800.0 PL=0
MOVL C01055 V=800.0 PL=0
MOVL C01056 V=800.0 PL=0
MOVL C01057 V=800.0 PL=0
MOVL C01058 V=800.0 PL=0
MOVL C01059 V=800.0 PL=0
MOVL C01060 V=800.0 PL=0
MOVL C01061 V=800.0 PL=0
MOVL C01062 V=800.0 PL=0
MOVL C01063 V=800.0 PL=0
MOVL C01064 V=800.0 PL=0
MOVL C01065 V=800.0 PL=0
MOVL C01066 V=800.0 PL=0
MOVL C01067 V=800.0 PL=0
MOVL C01068 V=800.0 PL=0
MOVL C01069 V=800.0 PL=0
MOVL C01070 V=800.0 PL=0
MOVL C01071 V=800.0 PL=0
MOVL C01072 V=800.0 PL=0
MOVL C01073 V=800.0 PL=0
MOVL C01074 V=800.0 PL=0
MOVL C01075 V=800.0 PL=0
MOVL C01076 V=800.0 PL=0
MOVL C01077 V=800.0 PL=0
MOVL C01078 V=800.0 PL=0
MOVL C01079 V=800.0 PL=0
MOVL C01080 V=800.0 PL=0
MOVL C01081 V=800.0 PL=0
MOVL C01082 V=800.0 PL=0
MOVL C01083 V=800.0 PL=0
MOVL C01084 V=800.0 PL=0
MOVL C01085 V=800.0 PL=0
MOVL C01086 V=800.0 PL=0
MOVL C01087 V=800.0 PL=0
MOVL C01088 V=800.0 PL=0
MOVL C01089 V=800.0 PL=0
MOVL C01090 V=800.0 PL=0
MOVL C01091 V=800.0 PL=0
MOVL C01092 V=800.0 PL=0
MOVL C01093 V=800.0 PL=0
MOVL C01094 V=800.0 PL=0
MOVL C01095 V=800.0 PL=0
MOVL C01096 V=800.0 PL=0
MOVL C01097 V=800.0 PL=0
MOVL C01098 V=800.0 PL=0
MOVL C01099 V=800.0 PL=0
MOVL C01100 V=800.0 PL=0
MOVL C01101 V=800.0 PL=0
MOVL C01102 V=800.0 PL=0
MOVL C01103 V=800.0 PL=0
MOVL C01104 V=800.0 PL=0
MOVL C01105 V=800.0 PL=0
MOVL C01106 V=800.0 PL=0
MOVL C01107 V=800.0 PL=0
MOVL C01108 V=800.0 PL=0
MOVL C01109 V=800.0 PL=0
MOVL C01110 V=800.0 PL=0
MOVL C01111 V=800.0 PL=0
MOVL C01112 V=800.0 PL=0
MOVL C01113 V=800.0 PL=0
MOVL C01114 V=800.0 PL=0
MOVL C01115 V=800.0 PL=0
MOVL C01116 V=800.0 PL=0
MOVL C01117 V=800.0 PL=0
MOVL C01118 V=800.0 PL=0
MOVL C01119 V=800.0 PL=0
MOVL C01120 V=800.0 PL=0
MOVL C01121 V=800.0 PL=0
MOVL C01122 V=800.0 PL=0
MOVL C01123 V=800.0 PL=0
MOVL C01124 V=800.0 PL=0
MOVL C01125 V=800.0 PL=0
MOVL C01126 V=800.0 PL=0
MOVL C01127 V=800.0 PL=0
MOVL C01128 V=800.0 PL=0
MOVL C01129 V=800.0 PL=0
MOVL C01130 V=800.0 PL=0
MOVL C01131 V=800.0 PL=0
MOVL C01132 V=800.0 PL=0
MOVL C01133 V=800.0 PL=0
MOVL C01134 V=800.0 PL=0
MOVL C01135 V=800.0 PL=0
MOVL C01136 V=800.0 PL=0
MOVL C01137 V=800.0 PL=0
MOVL C01138 V=800.0 PL=0
MOVL C01139 V=800.0 PL=0
MOVL C01140 V=800.0 PL=0
MOVL C01141 V=800.0 PL=0
MOVL C01142 V=800.0 PL=0
MOVL C01143 V=800.0 PL=0
MOVL C01144 V=800.0 PL=0
MOVL C01145 V=800.0 PL=0
MOVL C01146 V=800.0 PL=0
MOVL C01147 V=800.0 PL=0
MOVL C01148 V=800.0 PL=0
MOVL C01149 V=800.0 PL=0
MOVL C01150 V=800.0 PL=0
MOVL C01151 V=800.0 PL=0
MOVL C01152 V=800.0 PL=0
MOVL C01153 V=800.0 PL=0
MOVL C01154 V=800.0 PL=0
MOVL C01155 V=800.0 PL=0
MOVL C01156 V=800.0 PL=0
MOVL C01157 V=800.0 PL=0
MOVL C01158 V=800.0 PL=0
MOVL C01159 V=800.0 PL=0
MOVL C01160 V=800.0 PL=0
MOVL C01161 V=800.0 PL=0
MOVL C01162 V=800.0 PL=0
MOVL C01163 V=800.0 PL=0
MOVL C01164 V=800.0 PL=0
MOVL C01165 V=800.0 PL=0
MOVL C01166 V=800.0 PL=0
MOVL C01167 V=800.0 PL=0
MOVL C01168 V=800.0 PL=0
MOVL C01169 V=800.0 PL=0
MOVL C01170 V=800.0 PL=0
MOVL C01171 V=800.0 PL=0
MOVL C01172 V=800.0 PL=0
MOVL C01173 V=800.0 PL=0
MOVL C01174 V=800.0 PL=0
MOVL C01175 V=800.0 PL=0
MOVL C01176 V=800.0 PL=0
MOVL C01177 V=800.0 PL=0
MOVL C01178 V=800.0 PL=0
MOVL C01179 V=800.0 PL=0
MOVL C01180 V=800.0 PL=0
MOVL C01181 V=800.0 PL=0
MOVL C01182 V=800.0 PL=0
MOVL C01183 V=800.0 PL=0
MOVL C01184 V=800.0 PL=0
MOVL C01185 V=800.0 PL=0
MOVL C01186 V=800.0 PL=0
MOVL C01187 V=800.0 PL=0
MOVL C01188 V=800.0 PL=0
MOVL C01189 V=800.0 PL=0
MOVL C01190 V=800.0 PL=0
MOVL C01191 V=800.0 PL=0
MOVL C01192 V=800.0 PL=0
MOVL C01193 V=800.0 PL=0
MOVL C01194 V=800.0 PL=0
MOVL C01195 V=800.0 PL=0
MOVL C01196 V=800.0 PL=0
MOVL C01197 V=800.0 PL=0
MOVL C01198 V=800.0 PL=0
MOVL C01199 V=800.0 PL=0
MOVL C01200 V=800.0 PL=0
MOVL C01201 V=800.0 PL=0
MOVL C01202 V=800.0 PL=0
MOVL C01203 V=800.0 PL=0
MOVL C01204 V=800.0 PL=0
MOVL C01205 V=800.0 PL=0
MOVL C01206 V=800.0 PL=0
MOVL C01207 V=800.0 PL=0
MOVL C01208 V=800.0 PL=0
MOVL C01209 V=800.0 PL=0
MOVL C01210 V=800.0 PL=0
MOVL C01211 V=800.0 PL=0
MOVL C01212 V=800.0 PL=0
MOVL C01213 V=800.0 PL=0
MOVL C01214 V=800.0 PL=0
MOVL C01215 V=800.0 PL=0
MOVL C01216 V=800.0 PL=0
MOVL C01217 V=800.0 PL=0
MOVL C01218 V=800.0 PL=0
MOVL C01219 V=800.0 PL=0
MOVL C01220 V=800.0 PL=0
MOVL C01221 V=800.0 PL=0
MOVL C01222 V=800.0 PL=0
MOVL C01223 V=800.0 PL=0
MOVL C01224 V=800.0 PL=0
MOVL C01225 V=800.0 PL=0
MOVL C01226 V=800.0 PL=0
MOVL C01227 V=800.0 PL=0
MOVL C01228 V=800.0 PL=0
MOVL C01229 V=800.0 PL=0
MOVL C01230 V=800.0 PL=0
MOVL C01231 V=800.0 PL=0
MOVL C01232 V=800.0 PL=0
MOVL C01233 V=800.0 PL=0
MOVL C01234 V=800.0 PL=0
MOVL C01235 V=800.0 PL=0
MOVL C01236 V=800.0 PL=0
MOVL C01237 V=800.0 PL=0
MOVL C01238 V=800.0 PL=0
MOVL C01239 V=800.0 PL=0
MOVL C01240 V=800.0 PL=0
MOVL C01241 V=800.0 PL=0
MOVL C01242 V=800.0 PL=0
MOVL C01243 V=800.0 PL=0
MOVL C01244 V=800.0 PL=0
MOVL C01245 V=800.0 PL=0
MOVL C01246 V=800.0 PL=0
MOVL C01247 V=800.0 PL=0
MOVL C01248 V=800.0 PL=0
MOVL C01249 V=800.0 PL=0
MOVL C01250 V=800.0 PL=0
MOVL C01251 V=800.0 PL=0
MOVL C01252 V=800.0 PL=0
MOVL C01253 V=800.0 PL=0
MOVL C01254 V=800.0 PL=0
MOVL C01255 V=800.0 PL=0
MOVL C01256 V=800.0 PL=0
MOVL C01257 V=800.0 PL=0
MOVL C01258 V=800.0 PL=0
MOVL C01259 V=800.0 PL=0
MOVL C01260 V=800.0 PL=0
MOVL C01261 V=800.0 PL=0
MOVL C01262 V=800.0 PL=0
MOVL C01263 V=800.0 PL=0
MOVL C01264 V=800.0 PL=0
MOVL C01265 V=800.0 PL=0
MOVL C01266 V=800.0 PL=0
MOVL C01267 V=800.0 PL=0
MOVL C01268 V=800.0 PL=0
MOVL C01269 V=800.0 PL=0
MOVL C01270 V=800.0 PL=0
MOVL C01271 V=800.0 PL=0
MOVL C01272 V=800.0 PL=0
MOVL C01273 V=800.0 PL=0
MOVL C01274 V=800.0 PL=0
MOVL C01275 V=800.0 PL=0
MOVL C01276 V=800.0 PL=0
MOVL C01277 V=800.0 PL=0
MOVL C01278 V=800.0 PL=0
MOVL C01279 V=800.0 PL=0
MOVL C01280 V=800.0 PL=0
MOVL C01281 V=800.0 PL=0
MOVL C01282 V=800.0 PL=0
MOVL C01283 V=800.0 PL=0
MOVL C01284 V=800.0 PL=0
MOVL C01285 V=800.0 PL=0
MOVL C01286 V=800.0 PL=0
MOVL C01287 V=800.0 PL=0
MOVL C01288 V=800.0 PL=0
MOVL C01289 V=800.0 PL=0
MOVL C01290 V=800.0 PL=0
MOVL C01291 V=800.0 PL=0
MOVL C01292 V=800.0 PL=0
MOVL C01293 V=800.0 PL=0
MOVL C01294 V=800.0 PL=0
MOVL C01295 V=800.0 PL=0
MOVL C01296 V=800.0 PL=0
MOVL C01297 V=800.0 PL=0
MOVL C01298 V=800.0 PL=0
MOVL C01299 V=800.0 PL=0
MOVL C01300 V=800.0 PL=0
MOVL C01301 V=800.0 PL=0
MOVL C01302 V=800.0 PL=0
MOVL C01303 V=800.0 PL=0
MOVL C01304 V=800.0 PL=0
MOVL C01305 V=800.0 PL=0
MOVL C01306 V=800.0 PL=0
MOVL C01307 V=800.0 PL=0
MOVL C01308 V=800.0 PL=0
MOVL C01309 V=800.0 PL=0
MOVL C01310 V=800.0 PL=0
MOVL C01311 V=800.0 PL=0
MOVL C01312 V=800.0 PL=0
MOVL C01313 V=800.0 PL=0
MOVL C01314 V=800.0 PL=0
MOVL C01315 V=800.0 PL=0
MOVL C01316 V=800.0 PL=0
MOVL C01317 V=800.0 PL=0
MOVL C01318 V=800.0 PL=0
MOVL C01319 V=800.0 PL=0
MOVL C01320 V=800.0 PL=0
MOVL C01321 V=800.0 PL=0
MOVL C01322 V=800.0 PL=0
MOVL C01323 V=800.0 PL=0
MOVL C01324 V=800.0 PL=0
MOVL C01325 V=800.0 PL=0
MOVL C01326 V=800.0 PL=0
MOVL C01327 V=800.0 PL=0
MOVL C01328 V=800.0 PL=0
MOVL C01329 V=800.0 PL=0
MOVL C01330 V=800.0 PL=0
MOVL C01331 V=800.0 PL=0
MOVL C01332 V=800.0 PL=0
MOVL C01333 V=800.0 PL=0
MOVL C01334 V=800.0 PL=0
MOVL C01335 V=800.0 PL=0
MOVL C01336 V=800.0 PL=0
MOVL C01337 V=800.0 PL=0
MOVL C01338 V=800.0 PL=0
MOVL C01339 V=800.0 PL=0
MOVL C01340 V=800.0 PL=0
MOVL C01341 V=800.0 PL=0
MOVL C01342 V=800.0 PL=0
MOVL C01343 V=800.0 PL=0
MOVL C01344 V=800.0 PL=0
MOVL C01345 V=800.0 PL=0
MOVL C01346 V=800.0 PL=0
MOVL C01347 V=800.0 PL=0
MOVL C01348 V=800.0 PL=0
MOVL C01349 V=800.0 PL=0
MOVL C01350 V=800.0 PL=0
MOVL C01351 V=800.0 PL=0
MOVL C01352 V=800.0 PL=0
MOVL C01353 V=800.0 PL=0
MOVL C01354 V=800.0 PL=0
MOVL C01355 V=800.0 PL=0
MOVL C01356 V=800.0 PL=0
MOVL C01357 V=800.0 PL=0
MOVL C01358 V=800.0 PL=0
MOVL C01359 V=800.0 PL=0
MOVL C01360 V=800.0 PL=0
MOVL C01361 V=800.0 PL=0
MOVL C01362 V=800.0 PL=0
MOVL C01363 V=800.0 PL=0
MOVL C01364 V=800.0 PL=0
MOVL C01365 V=800.0 PL=0
MOVL C01366 V=800.0 PL=0
MOVL C01367 V=800.0 PL=0
MOVL C01368 V=800.0 PL=0
MOVL C01369 V=800.0 PL=0
MOVL C01370 V=800.0 PL=0
MOVL C01371 V=800.0 PL=0
MOVL C01372 V=800.0 PL=0
MOVL C01373 V=800.0 PL=0
MOVL C01374 V=800.0 PL=0
MOVL C01375 V=800.0 PL=0
MOVL C01376 V=800.0 PL=0
MOVL C01377 V=800.0 PL=0
MOVL C01378 V=800.0 PL=0
MOVL C01379 V=800.0 PL=0
MOVL C01380 V=800.0 PL=0
MOVL C01381 V=800.0 PL=0
MOVL C01382 V=800.0 PL=0
MOVL C01383 V=800.0 PL=0
MOVL C01384 V=800.0 PL=0
MOVL C01385 V=800.0 PL=0
MOVL C01386 V=800.0 PL=0
MOVL C01387 V=800.0 PL=0
MOVL C01388 V=800.0 PL=0
MOVL C01389 V=800.0 PL=0
MOVL C01390 V=800.0 PL=0
MOVL C01391 V=800.0 PL=0
MOVL C01392 V=800.0 PL=0
MOVL C01393 V=800.0 PL=0
MOVL C01394 V=800.0 PL=0
MOVL C01395 V=800.0 PL=0
MOVL C01396 V=800.0 PL=0
MOVL C01397 V=800.0 PL=0
MOVL C01398 V=800.0 PL=0
MOVL C01399 V=800.0 PL=0
MOVL C01400 V=800.0 PL=0
MOVL C01401 V=800.0 PL=0
MOVL C01402 V=800.0 PL=0
MOVL C01403 V=800.0 PL=0
MOVL C01404 V=800.0 PL=0
MOVL C01405 V=800.0 PL=0
MOVL C01406 V=800.0 PL=0
MOVL C01407 V=800.0 PL=0
MOVL C01408 V=800.0 PL=0
MOVL C01409 V=800.0 PL=0
MOVL C01410 V=800.0 PL=0
MOVL C01411 V=800.0 PL=0
MOVL C01412 V=800.0 PL=0
MOVL C01413 V=800.0 PL=0
MOVL C01414 V=800.0 PL=0
MOVL C01415 V=800.0 PL=0
MOVL C01416 V=800.0 PL=0
MOVL C01417 V=800.0 PL=0
MOVL C01418 V=800.0 PL=0
MOVL C01419 V=800.0 PL=0
MOVL C01420 V=800.0 PL=0
MOVL C01421 V=800.0 PL=0
MOVL C01422 V=800.0 PL=0
MOVL C01423 V=800.0 PL=0
MOVL C01424 V=800.0 PL=0
MOVL C01425 V=800.0 PL=0
MOVL C01426 V=800.0 PL=0
MOVL C01427 V=800.0 PL=0
MOVL C01428 V=800.0 PL=0
MOVL C01429 V=800.0 PL=0
MOVL C01430 V=800.0 PL=0
MOVL C01431 V=800.0 PL=0
MOVL C01432 V=800.0 PL=0
MOVL C01433 V=800.0 PL=0
MOVL C01434 V=800.0 PL=0
MOVL C01435 V=800.0 PL=0
MOVL C01436 V=800.0 PL=0
MOVL C01437 V=800.0 PL=0
MOVL C01438 V=800.0 PL=0
MOVL C01439 V=800.0 PL=0
MOVL C01440 V=800.0 PL=0
MOVL C01441 V=800.0 PL=0
MOVL C01442 V=800.0 PL=0
MOVL C01443 V=800.0 PL=0
MOVL C01444 V=800.0 PL=0
MOVL C01445 V=800.0 PL=0
MOVL C01446 V=800.0 PL=0
MOVL C01447 V=800.0 PL=0
MOVL C01448 V=800.0 PL=0
MOVL C01449 V=800.0 PL=0
MOVL C01450 V=800.0 PL=0
MOVL C01451 V=800.0 PL=0
MOVL C01452 V=800.0 PL=0
MOVL C01453 V=800.0 PL=0
MOVL C01454 V=800.0 PL=0
MOVL C01455 V=800.0 PL=0
MOVL C01456 V=800.0 PL=0
MOVL C01457 V=800.0 PL=0
MOVL C01458 V=800.0 PL=0
MOVL C01459 V=800.0 PL=0
MOVL C01460 V=800.0 PL=0
MOVL C01461 V=800.0 PL=0
MOVL C01462 V=800.0 PL=0
MOVL C01463 V=800.0 PL=0
MOVL C01464 V=800.0 PL=0
MOVL C01465 V=800.0 PL=0
MOVL C01466 V=800.0 PL=0
MOVL C01467 V=800.0 PL=0
MOVL C01468 V=800.0 PL=0
MOVL C01469 V=800.0 PL=0
MOVL C01470 V=800.0 PL=0
MOVL C01471 V=800.0 PL=0
MOVL C01472 V=800.0 PL=0
MOVL C01473 V=800.0 PL=0
MOVL C01474 V=800.0 PL=0
MOVL C01475 V=800.0 PL=0
MOVL C01476 V=800.0 PL=0
MOVL C01477 V=800.0 PL=0
MOVL C01478 V=800.0 PL=0
MOVL C01479 V=800.0 PL=0
MOVL C01480 V=800.0 PL=0
MOVL C01481 V=800.0 PL=0
MOVL C01482 V=800.0 PL=0
MOVL C01483 V=800.0 PL=0
MOVL C01484 V=800.0 PL=0
MOVL C01485 V=800.0 PL=0
MOVL C01486 V=800.0 PL=0
MOVL C01487 V=800.0 PL=0
MOVL C01488 V=800.0 PL=0
MOVL C01489 V=800.0 PL=0
MOVL C01490 V=800.0 PL=0
MOVL C01491 V=800.0 PL=0
MOVL C01492 V=800.0 PL=0
MOVL C01493 V=800.0 PL=0
MOVL C01494 V=800.0 PL=0
MOVL C01495 V=800.0 PL=0
MOVL C01496 V=800.0 PL=0
MOVL C01497 V=800.0 PL=0
MOVL C01498 V=800.0 PL=0
MOVL C01499 V=800.0 PL=0
MOVL C01500 V=800.0 PL=0
MOVL C01501 V=800.0 PL=0
MOVL C01502 V=800.0 PL=0
MOVL C01503 V=800.0 PL=0
MOVL C01504 V=800.0 PL=0
MOVL C01505 V=800.0 PL=0
MOVL C01506 V=800.0 PL=0
MOVL C01507 V=800.0 PL=0
MOVL C01508 V=800.0 PL=0
MOVL C01509 V=800.0 PL=0
MOVL C01510 V=800.0 PL=0
MOVL C01511 V=800.0 PL=0
MOVL C01512 V=800.0 PL=0
MOVL C01513 V=800.0 PL=0
MOVL C01514 V=800.0 PL=0
MOVL C01515 V=800.0 PL=0
MOVL C01516 V=800.0 PL=0
MOVL C01517 V=800.0 PL=0
MOVL C01518 V=800.0 PL=0
MOVL C01519 V=800.0 PL=0
MOVL C01520 V=800.0 PL=0
MOVL C01521 V=800.0 PL=0
MOVL C01522 V=800.0 PL=0
MOVL C01523 V=800.0 PL=0
MOVL C01524 V=800.0 PL=0
MOVL C01525 V=800.0 PL=0
MOVL C01526 V=800.0 PL=0
MOVL C01527 V=800.0 PL=0
MOVL C01528 V=800.0 PL=0
MOVL C01529 V=800.0 PL=0
MOVL C01530 V=800.0 PL=0
MOVL C01531 V=800.0 PL=0
MOVL C01532 V=800.0 PL=0
MOVL C01533 V=800.0 PL=0
MOVL C01534 V=800.0 PL=0
MOVL C01535 V=800.0 PL=0
MOVL C01536 V=800.0 PL=0
MOVL C01537 V=800.0 PL=0
MOVL C01538 V=800.0 PL=0
MOVL C01539 V=800.0 PL=0
MOVL C01540 V=800.0 PL=0
MOVL C01541 V=800.0 PL=0
MOVL C01542 V=800.0 PL=0
MOVL C01543 V=800.0 PL=0
MOVL C01544 V=800.0 PL=0
MOVL C01545 V=800.0 PL=0
MOVL C01546 V=800.0 PL=0
MOVL C01547 V=800.0 PL=0
MOVL C01548 V=800.0 PL=0
MOVL C01549 V=800.0 PL=0
MOVL C01550 V=800.0 PL=0
MOVL C01551 V=800.0 PL=0
MOVL C01552 V=800.0 PL=0
MOVL C01553 V=800.0 PL=0
MOVL C01554 V=800.0 PL=0
MOVL C01555 V=800.0 PL=0
MOVL C01556 V=800.0 PL=0
MOVL C01557 V=800.0 PL=0
MOVL C01558 V=800.0 PL=0
MOVL C01559 V=800.0 PL=0
MOVL C01560 V=800.0 PL=0
MOVL C01561 V=800.0 PL=0
MOVL C01562 V=800.0 PL=0
MOVL C01563 V=800.0 PL=0
MOVL C01564 V=800.0 PL=0
MOVL C01565 V=800.0 PL=0
MOVL C01566 V=800.0 PL=0
MOVL C01567 V=800.0 PL=0
MOVL C01568 V=800.0 PL=0
MOVL C01569 V=800.0 PL=0
MOVL C01570 V=800.0 PL=0
MOVL C01571 V=800.0 PL=0
MOVL C01572 V=800.0 PL=0
MOVL C01573 V=800.0 PL=0
MOVL C01574 V=800.0 PL=0
MOVL C01575 V=800.0 PL=0
MOVL C01576 V=800.0 PL=0
MOVL C01577 V=800.0 PL=0
MOVL C01578 V=800.0 PL=0
MOVL C01579 V=800.0 PL=0
MOVL C01580 V=800.0 PL=0
MOVL C01581 V=800.0 PL=0
MOVL C01582 V=800.0 PL=0
MOVL C01583 V=800.0 PL=0
MOVL C01584 V=800.0 PL=0
MOVL C01585 V=800.0 PL=0
MOVL C01586 V=800.0 PL=0
MOVL C01587 V=800.0 PL=0
MOVL C01588 V=800.0 PL=0
MOVL C01589 V=800.0 PL=0
MOVL C01590 V=800.0 PL=0
MOVL C01591 V=800.0 PL=0
MOVL C01592 V=800.0 PL=0
MOVL C01593 V=800.0 PL=0
MOVL C01594 V=800.0 PL=0
MOVL C01595 V=800.0 PL=0
MOVL C01596 V=800.0 PL=0
MOVL C01597 V=800.0 PL=0
MOVL C01598 V=800.0 PL=0
MOVL C01599 V=800.0 PL=0
MOVL C01600 V=800.0 PL=0
MOVL C01601 V=800.0 PL=0
MOVL C01602 V=800.0 PL=0
MOVL C01603 V=800.0 PL=0
MOVL C01604 V=800.0 PL=0
MOVL C01605 V=800.0 PL=0
MOVL C01606 V=800.0 PL=0
MOVL C01607 V=800.0 PL=0
MOVL C01608 V=800.0 PL=0
MOVL C01609 V=800.0 PL=0
MOVL C01610 V=800.0 PL=0
MOVL C01611 V=800.0 PL=0
MOVL C01612 V=800.0 PL=0
MOVL C01613 V=800.0 PL=0
MOVL C01614 V=800.0 PL=0
MOVL C01615 V=800.0 PL=0
MOVL C01616 V=800.0 PL=0
MOVL C01617 V=800.0 PL=0
MOVL C01618 V=800.0 PL=0
MOVL C01619 V=800.0 PL=0
MOVL C01620 V=800.0 PL=0
MOVL C01621 V=800.0 PL=0
MOVL C01622 V=800.0 PL=0
MOVL C01623 V=800.0 PL=0
MOVL C01624 V=800.0 PL=0
MOVL C01625 V=800.0 PL=0
MOVL C01626 V=800.0 PL=0
MOVL C01627 V=800.0 PL=0
MOVL C01628 V=800.0 PL=0
MOVL C01629 V=800.0 PL=0
MOVL C01630 V=800.0 PL=0
MOVL C01631 V=800.0 PL=0
MOVL C01632 V=800.0 PL=0
MOVL C01633 V=800.0 PL=0
MOVL C01634 V=800.0 PL=0
MOVL C01635 V=800.0 PL=0
MOVL C01636 V=800.0 PL=0
MOVL C01637 V=800.0 PL=0
MOVL C01638 V=800.0 PL=0
MOVL C01639 V=800.0 PL=0
MOVL C01640 V=800.0 PL=0
MOVL C01641 V=800.0 PL=0
MOVL C01642 V=800.0 PL=0
MOVL C01643 V=800.0 PL=0
MOVL C01644 V=800.0 PL=0
MOVL C01645 V=800.0 PL=0
MOVL C01646 V=800.0 PL=0
MOVL C01647 V=800.0 PL=0
MOVL C01648 V=800.0 PL=0
MOVL C01649 V=800.0 PL=0
MOVL C01650 V=800.0 PL=0
MOVL C01651 V=800.0 PL=0
MOVL C01652 V=800.0 PL=0
MOVL C01653 V=800.0 PL=0
MOVL C01654 V=800.0 PL=0
MOVL C01655 V=800.0 PL=0
MOVL C01656 V=800.0 PL=0
MOVL C01657 V=800.0 PL=0
MOVL C01658 V=800.0 PL=0
MOVL C01659 V=800.0 PL=0
MOVL C01660 V=800.0 PL=0
MOVL C01661 V=800.0 PL=0
MOVL C01662 V=800.0 PL=0
MOVL C01663 V=800.0 PL=0
MOVL C01664 V=800.0 PL=0
MOVL C01665 V=800.0 PL=0
MOVL C01666 V=800.0 PL=0
MOVL C01667 V=800.0 PL=0
MOVL C01668 V=800.0 PL=0
MOVL C01669 V=800.0 PL=0
MOVL C01670 V=800.0 PL=0
MOVL C01671 V=800.0 PL=0
MOVL C01672 V=800.0 PL=0
MOVL C01673 V=800.0 PL=0
MOVL C01674 V=800.0 PL=0
MOVL C01675 V=800.0 PL=0
MOVL C01676 V=800.0 PL=0
MOVL C01677 V=800.0 PL=0
MOVL C01678 V=800.0 PL=0
MOVL C01679 V=800.0 PL=0
MOVL C01680 V=800.0 PL=0
MOVL C01681 V=800.0 PL=0
MOVL C01682 V=800.0 PL=0
MOVL C01683 V=800.0 PL=0
MOVL C01684 V=800.0 PL=0
MOVL C01685 V=800.0 PL=0
MOVL C01686 V=800.0 PL=0
MOVL C01687 V=800.0 PL=0
MOVL C01688 V=800.0 PL=0
MOVL C01689 V=800.0 PL=0
MOVL C01690 V=800.0 PL=0
MOVL C01691 V=800.0 PL=0
MOVL C01692 V=800.0 PL=0
MOVL C01693 V=800.0 PL=0
MOVL C01694 V=800.0 PL=0
MOVL C01695 V=800.0 PL=0
MOVL C01696 V=800.0 PL=0
MOVL C01697 V=800.0 PL=0
MOVL C01698 V=800.0 PL=0
MOVL C01699 V=800.0 PL=0
MOVL C01700 V=800.0 PL=0
MOVL C01701 V=800.0 PL=0
MOVL C01702 V=800.0 PL=0
MOVL C01703 V=800.0 PL=0
MOVL C01704 V=800.0 PL=0
MOVL C01705 V=800.0 PL=0
MOVL C01706 V=800.0 PL=0
MOVL C01707 V=800.0 PL=0
MOVL C01708 V=800.0 PL=0
MOVL C01709 V=800.0 PL=0
MOVL C01710 V=800.0 PL=0
MOVL C01711 V=800.0 PL=0
MOVL C01712 V=800.0 PL=0
MOVL C01713 V=800.0 PL=0
MOVL C01714 V=800.0 PL=0
MOVL C01715 V=800.0 PL=0
MOVL C01716 V=800.0 PL=0
MOVL C01717 V=800.0 PL=0
MOVL C01718 V=800.0 PL=0
MOVL C01719 V=800.0 PL=0
MOVL C01720 V=800.0 PL=0
MOVL C01721 V=800.0 PL=0
MOVL C01722 V=800.0 PL=0
MOVL C01723 V=800.0 PL=0
MOVL C01724 V=800.0 PL=0
MOVL C01725 V=800.0 PL=0
MOVL C01726 V=800.0 PL=0
MOVL C01727 V=800.0 PL=0
MOVL C01728 V=800.0 PL=0
MOVL C01729 V=800.0 PL=0
MOVL C01730 V=800.0 PL=0
MOVL C01731 V=800.0 PL=0
MOVL C01732 V=800.0 PL=0
MOVL C01733 V=800.0 PL=0
MOVL C01734 V=800.0 PL=0
MOVL C01735 V=800.0 PL=0
MOVL C01736 V=800.0 PL=0
MOVL C01737 V=800.0 PL=0
MOVL C01738 V=800.0 PL=0
MOVL C01739 V=800.0 PL=0
MOVL C01740 V=800.0 PL=0
MOVL C01741 V=800.0 PL=0
MOVL C01742 V=800.0 PL=0
MOVL C01743 V=800.0 PL=0
MOVL C01744 V=800.0 PL=0
MOVL C01745 V=800.0 PL=0
MOVL C01746 V=800.0 PL=0
MOVL C01747 V=800.0 PL=0
MOVL C01748 V=800.0 PL=0
MOVL C01749 V=800.0 PL=0
MOVL C01750 V=800.0 PL=0
MOVL C01751 V=800.0 PL=0
MOVL C01752 V=800.0 PL=0
MOVL C01753 V=800.0 PL=0
MOVL C01754 V=800.0 PL=0
MOVL C01755 V=800.0 PL=0
MOVL C01756 V=800.0 PL=0
MOVL C01757 V=800.0 PL=0
MOVL C01758 V=800.0 PL=0
MOVL C01759 V=800.0 PL=0
MOVL C01760 V=800.0 PL=0
MOVL C01761 V=800.0 PL=0
MOVL C01762 V=800.0 PL=0
MOVL C01763 V=800.0 PL=0
MOVL C01764 V=800.0 PL=0
MOVL C01765 V=800.0 PL=0
MOVL C01766 V=800.0 PL=0
MOVL C01767 V=800.0 PL=0
MOVL C01768 V=800.0 PL=0
MOVL C01769 V=800.0 PL=0
MOVL C01770 V=800.0 PL=0
MOVL C01771 V=800.0 PL=0
MOVL C01772 V=800.0 PL=0
MOVL C01773 V=800.0 PL=0
MOVL C01774 V=800.0 PL=0
MOVL C01775 V=800.0 PL=0
MOVL C01776 V=800.0 PL=0
MOVL C01777 V=800.0 PL=0
MOVL C01778 V=800.0 PL=0
MOVL C01779 V=800.0 PL=0
MOVL C01780 V=800.0 PL=0
MOVL C01781 V=800.0 PL=0
MOVL C01782 V=800.0 PL=0
MOVL C01783 V=800.0 PL=0
MOVL C01784 V=800.0 PL=0
MOVL C01785 V=800.0 PL=0
MOVL C01786 V=800.0 PL=0
MOVL C01787 V=800.0 PL=0
MOVL C01788 V=800.0 PL=0
MOVL C01789 V=800.0 PL=0
MOVL C01790 V=800.0 PL=0
MOVL C01791 V=800.0 PL=0
MOVL C01792 V=800.0 PL=0
MOVL C01793 V=800.0 PL=0
MOVL C01794 V=800.0 PL=0
MOVL C01795 V=800.0 PL=0
MOVL C01796 V=800.0 PL=0
MOVL C01797 V=800.0 PL=0
MOVL C01798 V=800.0 PL=0
MOVL C01799 V=800.0 PL=0
MOVL C01800 V=800.0 PL=0
MOVL C01801 V=800.0 PL=0
MOVL C01802 V=800.0 PL=0
MOVL C01803 V=800.0 PL=0
MOVL C01804 V=800.0 PL=0
MOVL C01805 V=800.0 PL=0
MOVL C01806 V=800.0 PL=0
MOVL C01807 V=800.0 PL=0
MOVL C01808 V=800.0 PL=0
MOVL C01809 V=800.0 PL=0
MOVL C01810 V=800.0 PL=0
MOVL C01811 V=800.0 PL=0
MOVL C01812 V=800.0 PL=0
MOVL C01813 V=800.0 PL=0
MOVL C01814 V=800.0 PL=0
MOVL C01815 V=800.0 PL=0
MOVL C01816 V=800.0 PL=0
MOVL C01817 V=800.0 PL=0
MOVL C01818 V=800.0 PL=0
MOVL C01819 V=800.0 PL=0
MOVL C01820 V=800.0 PL=0
MOVL C01821 V=800.0 PL=0
MOVL C01822 V=800.0 PL=0
MOVL C01823 V=800.0 PL=0
MOVL C01824 V=800.0 PL=0
MOVL C01825 V=800.0 PL=0
MOVL C01826 V=800.0 PL=0
MOVL C01827 V=800.0 PL=0
MOVL C01828 V=800.0 PL=0
MOVL C01829 V=800.0 PL=0
MOVL C01830 V=800.0 PL=0
MOVL C01831 V=800.0 PL=0
MOVL C01832 V=800.0 PL=0
MOVL C01833 V=800.0 PL=0
MOVL C01834 V=800.0 PL=0
MOVL C01835 V=800.0 PL=0
MOVL C01836 V=800.0 PL=0
MOVL C01837 V=800.0 PL=0
MOVL C01838 V=800.0 PL=0
MOVL C01839 V=800.0 PL=0
MOVL C01840 V=800.0 PL=0
MOVL C01841 V=800.0 PL=0
MOVL C01842 V=800.0 PL=0
MOVL C01843 V=800.0 PL=0
MOVL C01844 V=800.0 PL=0
MOVL C01845 V=800.0 PL=0
MOVL C01846 V=800.0 PL=0
MOVL C01847 V=800.0 PL=0
MOVL C01848 V=800.0 PL=0
MOVL C01849 V=800.0 PL=0
MOVL C01850 V=800.0 PL=0
MOVL C01851 V=800.0 PL=0
MOVL C01852 V=800.0 PL=0
MOVL C01853 V=800.0 PL=0
MOVL C01854 V=800.0 PL=0
MOVL C01855 V=800.0 PL=0
MOVL C01856 V=800.0 PL=0
MOVL C01857 V=800.0 PL=0
MOVL C01858 V=800.0 PL=0
MOVL C01859 V=800.0 PL=0
MOVL C01860 V=800.0 PL=0
MOVL C01861 V=800.0 PL=0
MOVL C01862 V=800.0 PL=0
MOVL C01863 V=800.0 PL=0
MOVL C01864 V=800.0 PL=0
MOVL C01865 V=800.0 PL=0
MOVL C01866 V=800.0 PL=0
MOVL C01867 V=800.0 PL=0
MOVL C01868 V=800.0 PL=0
MOVL C01869 V=800.0 PL=0
MOVL C01870 V=800.0 PL=0
MOVL C01871 V=800.0 PL=0
MOVL C01872 V=800.0 PL=0
MOVL C01873 V=800.0 PL=0
MOVL C01874 V=800.0 PL=0
MOVL C01875 V=800.0 PL=0
MOVL C01876 V=800.0 PL=0
MOVL C01877 V=800.0 PL=0
MOVL C01878 V=800.0 PL=0
MOVL C01879 V=800.0 PL=0
MOVL C01880 V=800.0 PL=0
MOVL C01881 V=800.0 PL=0
MOVL C01882 V=800.0 PL=0
MOVL C01883 V=800.0 PL=0
MOVL C01884 V=800.0 PL=0
MOVL C01885 V=800.0 PL=0
MOVL C01886 V=800.0 PL=0
MOVL C01887 V=800.0 PL=0
MOVL C01888 V=800.0 PL=0
MOVL C01889 V=800.0 PL=0
MOVL C01890 V=800.0 PL=0
MOVL C01891 V=800.0 PL=0
MOVL C01892 V=800.0 PL=0
MOVL C01893 V=800.0 PL=0
MOVL C01894 V=800.0 PL=0
MOVL C01895 V=800.0 PL=0
MOVL C01896 V=800.0 PL=0
MOVL C01897 V=800.0 PL=0
MOVL C01898 V=800.0 PL=0
MOVL C01899 V=800.0 PL=0
MOVL C01900 V=800.0 PL=0
MOVL C01901 V=800.0 PL=0
MOVL C01902 V=800.0 PL=0
MOVL C01903 V=800.0 PL=0
MOVL C01904 V=800.0 PL=0
MOVL C01905 V=800.0 PL=0
MOVL C01906 V=800.0 PL=0
MOVL C01907 V=800.0 PL=0
MOVL C01908 V=800.0 PL=0
MOVL C01909 V=800.0 PL=0
MOVL C01910 V=800.0 PL=0
MOVL C01911 V=800.0 PL=0
MOVL C01912 V=800.0 PL=0
MOVL C01913 V=800.0 PL=0
MOVL C01914 V=800.0 PL=0
MOVL C01915 V=800.0 PL=0
MOVL C01916 V=800.0 PL=0
MOVL C01917 V=800.0 PL=0
MOVL C01918 V=800.0 PL=0
MOVL C01919 V=800.0 PL=0
MOVL C01920 V=800.0 PL=0
MOVL C01921 V=800.0 PL=0
MOVL C01922 V=800.0 PL=0
MOVL C01923 V=800.0 PL=0
MOVL C01924 V=800.0 PL=0
MOVL C01925 V=800.0 PL=0
MOVL C01926 V=800.0 PL=0
MOVL C01927 V=800.0 PL=0
MOVL C01928 V=800.0 PL=0
MOVL C01929 V=800.0 PL=0
MOVL C01930 V=800.0 PL=0
MOVL C01931 V=800.0 PL=0
MOVL C01932 V=800.0 PL=0
MOVL C01933 V=800.0 PL=0
MOVL C01934 V=800.0 PL=0
MOVL C01935 V=800.0 PL=0
MOVL C01936 V=800.0 PL=0
MOVL C01937 V=800.0 PL=0
MOVL C01938 V=800.0 PL=0
MOVL C01939 V=800.0 PL=0
MOVL C01940 V=800.0 PL=0
MOVL C01941 V=800.0 PL=0
MOVL C01942 V=800.0 PL=0
MOVL C01943 V=800.0 PL=0
MOVL C01944 V=800.0 PL=0
MOVL C01945 V=800.0 PL=0
MOVL C01946 V=800.0 PL=0
MOVL C01947 V=800.0 PL=0
MOVL C01948 V=800.0 PL=0
MOVL C01949 V=800.0 PL=0
MOVL C01950 V=800.0 PL=0
MOVL C01951 V=800.0 PL=0
MOVL C01952 V=800.0 PL=0
MOVL C01953 V=800.0 PL=0
MOVL C01954 V=800.0 PL=0
MOVL C01955 V=800.0 PL=0
MOVL C01956 V=800.0 PL=0
MOVL C01957 V=800.0 PL=0
MOVL C01958 V=800.0 PL=0
MOVL C01959 V=800.0 PL=0
MOVL C01960 V=800.0 PL=0
MOVL C01961 V=800.0 PL=0
MOVL C01962 V=800.0 PL=0
MOVL C01963 V=800.0 PL=0
MOVL C01964 V=800.0 PL=0
MOVL C01965 V=800.0 PL=0
MOVL C01966 V=800.0 PL=0
MOVL C01967 V=800.0 PL=0
MOVL C01968 V=800.0 PL=0
MOVL C01969 V=800.0 PL=0
MOVL C01970 V=800.0 PL=0
MOVL C01971 V=800.0 PL=0
MOVL C01972 V=800.0 PL=0
MOVL C01973 V=800.0 PL=0
MOVL C01974 V=800.0 PL=0
MOVL C01975 V=800.0 PL=0
MOVL C01976 V=800.0 PL=0
MOVL C01977 V=800.0 PL=0
MOVL C01978 V=800.0 PL=0
MOVL C01979 V=800.0 PL=0
MOVL C01980 V=800.0 PL=0
MOVL C01981 V=800.0 PL=0
MOVL C01982 V=800.0 PL=0
MOVL C01983 V=800.0 PL=0
MOVL C01984 V=800.0 PL=0
MOVL C01985 V=800.0 PL=0
MOVL C01986 V=800.0 PL=0
MOVL C01987 V=800.0 PL=0
MOVL C01988 V=800.0 PL=0
MOVL C01989 V=800.0 PL=0
MOVL C01990 V=800.0 PL=0
MOVL C01991 V=800.0 PL=0
MOVL C01992 V=800.0 PL=0
MOVL C01993 V=800.0 PL=0
MOVL C01994 V=800.0 PL=0
MOVL C01995 V=800.0 PL=0
MOVL C01996 V=800.0 PL=0
MOVL C01997 V=800.0 PL=0
MOVL C01998 V=800.0 PL=0
MOVL C01999 V=800.0 PL=0
MOVL C02000 V=800.0 PL=0
MOVL C02001 V=800.0 PL=0
MOVL C02002 V=800.0 PL=0
MOVL C02003 V=800.0 PL=0
MOVL C02004 V=800.0 PL=0
MOVL C02005 V=800.0 PL=0
MOVL C02006 V=800.0 PL=0
MOVL C02007 V=800.0 PL=0
MOVL C02008 V=800.0 PL=0
MOVL C02009 V=800.0 PL=0
MOVL C02010 V=800.0 PL=0
MOVL C02011 V=800.0 PL=0
MOVL C02012 V=800.0 PL=0
MOVL C02013 V=800.0 PL=0
MOVL C02014 V=800.0 PL=0
MOVL C02015 V=800.0 PL=0
MOVL C02016 V=800.0 PL=0
MOVL C02017 V=800.0 PL=0
MOVL C02018 V=800.0 PL=0
MOVL C02019 V=800.0 PL=0
MOVL C02020 V=800.0 PL=0
MOVL C02021 V=800.0 PL=0
MOVL C02022 V=800.0 PL=0
MOVL C02023 V=800.0 PL=0
MOVL C02024 V=800.0 PL=0
MOVL C02025 V=800.0 PL=0
MOVL C02026 V=800.0 PL=0
MOVL C02027 V=800.0 PL=0
MOVL C02028 V=800.0 PL=0
MOVL C02029 V=800.0 PL=0
MOVL C02030 V=800.0 PL=0
MOVL C02031 V=800.0 PL=0
MOVL C02032 V=800.0 PL=0
MOVL C02033 V=800.0 PL=0
MOVL C02034 V=800.0 PL=0
MOVL C02035 V=800.0 PL=0
MOVL C02036 V=800.0 PL=0
MOVL C02037 V=800.0 PL=0
MOVL C02038 V=800.0 PL=0
MOVL C02039 V=800.0 PL=0
MOVL C02040 V=800.0 PL=0
MOVL C02041 V=800.0 PL=0
MOVL C02042 V=800.0 PL=0
MOVL C02043 V=800.0 PL=0
MOVL C02044 V=800.0 PL=0
MOVL C02045 V=800.0 PL=0
MOVL C02046 V=800.0 PL=0
MOVL C02047 V=800.0 PL=0
MOVL C02048 V=800.0 PL=0
MOVL C02049 V=800.0 PL=0
MOVL C02050 V=800.0 PL=0
MOVL C02051 V=800.0 PL=0
MOVL C02052 V=800.0 PL=0
MOVL C02053 V=800.0 PL=0
MOVL C02054 V=800.0 PL=0
MOVL C02055 V=800.0 PL=0
MOVL C02056 V=800.0 PL=0
MOVL C02057 V=800.0 PL=0
MOVL C02058 V=800.0 PL=0
MOVL C02059 V=800.0 PL=0
MOVL C02060 V=800.0 PL=0
MOVL C02061 V=800.0 PL=0
MOVL C02062 V=800.0 PL=0
MOVL C02063 V=800.0 PL=0
MOVL C02064 V=800.0 PL=0
MOVL C02065 V=800.0 PL=0
MOVL C02066 V=800.0 PL=0
MOVL C02067 V=800.0 PL=0
MOVL C02068 V=800.0 PL=0
MOVL C02069 V=800.0 PL=0
MOVL C02070 V=800.0 PL=0
MOVL C02071 V=800.0 PL=0
MOVL C02072 V=800.0 PL=0
MOVL C02073 V=800.0 PL=0
MOVL C02074 V=800.0 PL=0
MOVL C02075 V=800.0 PL=0
MOVL C02076 V=800.0 PL=0
MOVL C02077 V=800.0 PL=0
MOVL C02078 V=800.0 PL=0
MOVL C02079 V=800.0 PL=0
MOVL C02080 V=800.0 PL=0
MOVL C02081 V=800.0 PL=0
MOVL C02082 V=800.0 PL=0
MOVL C02083 V=800.0 PL=0
MOVL C02084 V=800.0 PL=0
MOVL C02085 V=800.0 PL=0
MOVL C02086 V=800.0 PL=0
MOVL C02087 V=800.0 PL=0
MOVL C02088 V=800.0 PL=0
MOVL C02089 V=800.0 PL=0
MOVL C02090 V=800.0 PL=0
MOVL C02091 V=800.0 PL=0
MOVL C02092 V=800.0 PL=0
MOVL C02093 V=800.0 PL=0
MOVL C02094 V=800.0 PL=0
MOVL C02095 V=800.0 PL=0
MOVL C02096 V=800.0 PL=0
MOVL C02097 V=800.0 PL=0
MOVL C02098 V=800.0 PL=0
MOVL C02099 V=800.0 PL=0
MOVL C02100 V=800.0 PL=0
MOVL C02101 V=800.0 PL=0
MOVL C02102 V=800.0 PL=0
MOVL C02103 V=800.0 PL=0
MOVL C02104 V=800.0 PL=0
MOVL C02105 V=800.0 PL=0
MOVL C02106 V=800.0 PL=0
MOVL C02107 V=800.0 PL=0
MOVL C02108 V=800.0 PL=0
MOVL C02109 V=800.0 PL=0
MOVL C02110 V=800.0 PL=0
MOVL C02111 V=800.0 PL=0
MOVL C02112 V=800.0 PL=0
MOVL C02113 V=800.0 PL=0
MOVL C02114 V=800.0 PL=0
